	81200:
			TON_DelayTransMove.IN := false;
			IF 	LowerConveyor.InStopped THEN
				tonTimeOut.IN:=FALSE;
				uiExecutingStep:=99000;
			END_IF
			tonTimeOut.IN:=TRUE;
			IF tonTimeOut.Q=TRUE THEN
				strStatus :='Stop conveyor timeout';
				_Error:=TRUE;
			END_IF		
					
    99000: // process done
          Status    := 'Process completed';
      	  _Executed := TRUE;
END_CASE
IF _Executed THEN
    eState := STATE_DONE;
ELSIF _Error THEN
//	FUN_UniqueErrorCodeGenerator(iErrorID := ErrorID,UinqueErrorCode=>_UniqueErrorCode);
    eState := STATE_ERROR;
ELSIF NOT Execute THEN
    eState := STATE_RESETTING;
END_IF
IF _Abort OR Abort THEN
//	FUN_UniqueErrorCodeGenerator(iErrorID := ErrorID,UinqueErrorCode=>_UniqueErrorCode);
	eSTATE:=STATE_ABORTING;
END_IF
END_METHOD

METHOD  M_STATE_RESETTING
VAR_INPUT
END_VAR
Error :=FALSE;
Done :=FALSE;
Busy := FALSE;


CASE uiResettingStep OF
	
	0:
		tonTimeOut.IN:=FALSE;
		TON_DelayTransMove.IN :=FALSE;
		Robot.M_ResetAllCommand();
		Robot.M_ResetRobotAbsMove(TRUE,TRUE);
		uiResettingStep:=100;
		
	100:
	
		LowerConveyor.M_MotorStop();	
		uiResettingStep:=9999;
	9999:
		_ResetCompleted:=TRUE;
END_CASE
IF _ResetCompleted THEN
	eSTATE:=STATE_DORMANT;
END_IF
END_METHOD

END_FUNCTION_BLOCK

// ---- Library/20_MachineUnits/21_StorageArea/Old_version_Service/FB_WareHouseInnerPickToRoundBeltBatch_Old.TcPOU
// ═══════════════════════════════════════════════════════════════════════════
// FB_WareHouseInnerPickToRoundBeltBatch
// 倉儲內層取盒放圓帶 — 批次服務 FB
// ═══════════════════════════════════════════════════════════════════════════
//
// 【用途】
// 管理最多 40 筆「從倉儲內層取盒放上圓帶」流程,每筆由 FB_WareHouseInnerPickToRoundBelt
// 逐筆執行。批次流程由 C# HMI 透過 ADS 寫入 BatchInfo 結構觸發,PLC 端負責
// 驗證資料、迭代處理、handshake 同步動作紀錄給 C#。
//
// 【設計模式】
// 參照 FB_AllocateMoveAutoBatchMode,以「單筆 FB 內嵌 + 批次迭代」架構:
//   1. 收到 Execute → 驗證整批資料安全 (M_ValidateBatchData)
//   2. 迭代 FlowInfo[0..NrOfFlow-1]
//   3. 跳過無效項 (ID = -1 或 A/B 爪皆 NoWork)
//   4. 對每筆有效流程配置並啟動 fbSingleFlow,等其完成/失敗
//   5. 完成後記錄 WorkedID 供 HMI/C# 回報
//   6. 跨迭代 handshake 清理,確保 C# 看到每筆 FeedBack 上升緣
//
// 【FeedBack / ReadComplete 握手協定】(關鍵,跨迭代正確性依賴)
// 每筆 fbSingleFlow 完成時:
//   PLC:   step 99000 → FeedBack := TRUE (通知 C# 陣列可讀)
//   C#:    收到 FeedBack=TRUE → 讀 ActionRecords → set ReadComplete=TRUE
//   PLC:   step 99100 看 ReadComplete=TRUE → 清 FeedBack → 進 DONE
//   C#:    應在看到 FeedBack=FALSE 時清 ReadComplete=FALSE (維持協定)
// 本 Batch FB 為了防 C# 忘記清 ReadComplete 造成下一迭代 skip handshake,
// 在 Step 100 (新迭代開始) 與 Step 300 (迭代結束) 強制清 BatchInfo.ReadComplete。
//
// 【資料安全約束】
// M_ValidateBatchData 在 Step 0 首次進入時呼叫,檢查:
//   - 每個 Work clamp 的 Station 不可為 Undefined
//   - 所有 Work clamp 的 (Station, ReloadCarrier) 不可重複 (同 flow A/B 兩爪也算)
// 違規 → Error + uiResumeStep:=0 (不可續做,需 C# 修正資料重來)
//
// 【Resume / Pause】
// Resume: 錯誤/逾時後 C# 按 Reset → RESETTING 等 fbSingleFlow 回 DORMANT
//         → 若 _bRetry 直接回 EXECUTING 從 uiResumeStep 繼續
//         uiResumeStep 映射固定為 100 (重新配置+啟動 fbSingleFlow),因 abort
//         過程會清掉 fbSingleFlow 內部狀態,不能回原 step 200
// Pause:  僅在「迭代邊界」生效 (step 0 或 310),不中斷單筆流程
//         危險區段 (100~300) 繼續跑到下個邊界才凍結
//
// Create Date : 2026/04/01
// Owner       : Copilot
// ═══════════════════════════════════════════════════════════════════════════

FUNCTION_BLOCK FB_WareHouseInnerPickToRoundBeltBatch_Old EXTENDS FB_ObjectBase_V2 IMPLEMENTS IBasicElement

VAR_INPUT
	// ----- 外部資源參照 (由上層 FB_StorageArea 綁定) -----
	Robot			: REFERENCE TO FB_FanucRobot_Basic_V2;	// 倉儲區 Fanuc 手臂 (取放動作執行者)
	RoundBelt		: REFERENCE TO FB_RoundBeltService;		// 圓帶服務 (目的地,換區偵測)
	WareHouse		: REFERENCE TO FB_WareHouse;				// 倉儲 FB (ReloadBox / FeedInBox)
	Input			: ST_InputTable;						// IO 輸入表 (sensor 等)

	// ----- 批次資料 (C# HMI ↔ PLC 介面) -----
	// BatchInfo 由 C# 透過 ADS 寫入;PLC 讀 FlowInfo[] 並回寫 WorkedID / ActionRecords
	BatchInfo		: REFERENCE TO ST_WareHouseInnerPickBatch;

	Stop			: BOOL;									// 外部停止信號 (DORMANT 時阻擋 Execute 觸發)
END_VAR

VAR_OUTPUT
	// 無額外 output — 完成/錯誤/忙碌狀態透過 BatchInfo.HandShake 回傳 C#
END_VAR

VAR
	// ----- 狀態與錯誤追蹤 -----
	strStatus			: STRING;			// 當前狀態/錯誤描述 (顯示給 HMI)
	tonTimeOut			: TON;				// Per-iteration 逾時計時器 (PT=600s, step 310 推進時重置)
	_UniqueErrorCode	: STRING;			// 錯誤代碼 (E_NOT_AUTO_MODE / E_BATCH_TIMEOUT / E_FLOW_FAILED /
											// E_STATION_UNDEFINED / E_DUPLICATE_TARGET)
	uiResumeStep		: UDINT := 0;		// 續做點步序 (0 = 不可續做, 其他 = RESETTING retry 回此 step)
	_bRetry				: BOOL;				// 續做旗標 (ABORTED → RESETTING → EXECUTING 路徑標記)

	// ----- 批次迭代控制 -----
	iProcessingIndex	: INT := 0;		// 當前處理的流程索引 (0..NrOfFlow-1)
										// 注意: 續做時保留不歸零 (僅 DORMANT 清),保證從中斷點繼續
	CurrentFlow			: ST_WareHouseInnerPickFlowInfo;	// 當前流程資料快取 (避免 C# 改寫中讀取)

	// ----- 內嵌單筆 FB -----
	// 每筆流程都透過這個實例執行;Step 100 配置參照+啟動,Step 310 等其回到 DORMANT
	fbSingleFlow		: FB_WareHouseInnerPickToRoundBelt;
	_bSingleFlowStarted	: BOOL;		// 追蹤 fbSingleFlow 是否有待清理的執行狀態 (用於 ABORTING)
END_VAR

// ============================================================
// 執行順序: input piping → A00 → A10 → output piping
// 讓 state machine 內的 fbSingleFlow() 看到當前 scan 的 C# 輸入
// (ReadComplete),避免 1 scan 延遲
// ============================================================

// 1. Input piping: C# → fbSingleFlow (在 state machine 前)
IF __ISVALIDREF(BatchInfo) THEN
	fbSingleFlow.ReadComplete := BatchInfo.ReadComplete;
END_IF

// 2. Timer PT setup
A00_BasicUnits();

// 3. State machine (含 fbSingleFlow() 呼叫)
SUPER^.A10_StateControl();

// 4. Output piping: fbSingleFlow → C#
IF __ISVALIDREF(BatchInfo) THEN
	BatchInfo.ActionRecords := fbSingleFlow.ActionRecords;
	BatchInfo.ActionIndex := fbSingleFlow.ActionIndex;
	BatchInfo.FeedBack := fbSingleFlow.FeedBack;
	BatchInfo.HandShake.Done := Done;
	BatchInfo.HandShake.Busy := Busy;
	BatchInfo.HandShake.Error := Error;
END_IF
fbSingleFlow (Input := Input);

ACTION A00_BasicUnits:
// 每單筆流程上限 (per-iteration timeout,由 EXECUTING step 310 重置)
// 最多 40 筆 x 600s 單筆 = 6.7hr 批次上限足夠
tonTimeOut(PT := T#900S);
END_ACTION

// 尋找下一筆有效流程
// 從 iProcessingIndex 開始往後掃描 BatchInfo.FlowInfo[]
// 有效條件: ID <> -1 且至少一爪為 Work
// 無效流程自動跳過並記錄 WorkedID
// 回傳 TRUE = 找到有效流程 (iProcessingIndex 已更新), FALSE = 全部完成
METHOD M_FindNextValidFlow : BOOL
VAR_INPUT
END_VAR
VAR
	i		: INT;
	bValid	: BOOL;
END_VAR
IF NOT __ISVALIDREF(BatchInfo) THEN
	M_FindNextValidFlow := FALSE;
	RETURN;
END_IF

IF BatchInfo.NrOfFlow = 0 THEN
	M_FindNextValidFlow := FALSE;
	RETURN;
END_IF

FOR i := iProcessingIndex TO UINT_TO_INT(BatchInfo.NrOfFlow) - 1 BY 1 DO
	bValid := FALSE;

	// 檢查 flow 是否有效 (ID 不為 -1)
	IF BatchInfo.FlowInfo[i].ID <> -1 THEN
		// 檢查是否至少一爪有 Work 行為
		IF BatchInfo.FlowInfo[i].ClampA_Setting.Behavior = E_ClampWork.Work
		OR BatchInfo.FlowInfo[i].ClampB_Setting.Behavior = E_ClampWork.Work THEN
			bValid := TRUE;
		END_IF
	END_IF

	IF bValid THEN
		iProcessingIndex := i;
		CurrentFlow := BatchInfo.FlowInfo[i];
		M_FindNextValidFlow := TRUE;
		RETURN;
	ELSE
		// 標記跳過的 flow 為已處理
		BatchInfo.WorkedID[i] := BatchInfo.FlowInfo[i].ID;
	END_IF
END_FOR

// 沒有更多有效流程
M_FindNextValidFlow := FALSE;
END_METHOD

// ───────────────────────────────────────────────────────────
// M_STATE_ABORTED — 已中止 (可續做錯誤)
// ───────────────────────────────────────────────────────────
// 進入條件:
//   M_STATE_ABORTING 完成清理 (_AbortCompleted=TRUE) 後進入
//
// 特性:
//   - 顯示 Aborted=TRUE + Error=TRUE + strStatus
//   - 等待 C# 透過 BatchInfo.HandShake.Reset 觸發續做或重來
//
// Reset 行為:
//   - uiResumeStep > 0 → 設 _bRetry, uiExecutingStep := uiResumeStep
//                        RESETTING 會等 fbSingleFlow 回 DORMANT 後直接跳 EXECUTING
//                        (從中斷點續做,保留 iProcessingIndex)
//   - uiResumeStep = 0 → 單純 RESETTING → DORMANT,下次 Execute 從頭跑
METHOD M_STATE_ABORTED
VAR_INPUT
END_VAR
Busy := FALSE;
Aborted := TRUE;
Error := TRUE;
Status := strStatus;
_AbortCompleted := FALSE;
uiAbortingStep :=0;

// Support retry/resume on Reset
IF __ISVALIDREF(BatchInfo) THEN
	IF BatchInfo.HandShake.Reset THEN
		IF uiResumeStep > 0 THEN
			uiExecutingStep := uiResumeStep;
			_bRetry := TRUE;
		END_IF
		eState := STATE_RESETTING;
	END_IF
END_IF
END_METHOD

// ───────────────────────────────────────────────────────────
// M_STATE_ABORTING — 中止流程
// ───────────────────────────────────────────────────────────
// 職責:
//   把正在執行的 fbSingleFlow 中止,等其自身 ABORTING → ABORTED
//   跑完後設 _AbortCompleted 進入 STATE_ABORTED。
//   fbSingleFlow 的 ABORTING 內部會處理 Robot/WareHouse/RoundBelt 的資源釋放。
//
// 進入條件:
//   M_STATE_EXECUTING 設 _Abort := TRUE 時觸發
//   (timeout, 單筆流程失敗, Auto mode 脫離等)
//
// 步序:
//   0:    若 _bSingleFlowStarted=TRUE → 發送 fbSingleFlow.Abort := TRUE, 跳 100
//         (若單筆 FB 尚未啟動過,直接跳 9999 略過等待)
//   100:  每 cycle 呼叫 fbSingleFlow() 推進其內部中止狀態機
//         等待條件 (任一滿足): 未啟動 / fbSingleFlow.Aborted / fbSingleFlow 不忙碌
//         → 清 fbSingleFlow.Abort := FALSE, 跳 9999
//   9999: _AbortCompleted := TRUE → base class 轉入 STATE_ABORTED
//
// 注意:
//   iProcessingIndex 不在此清除 (保留供續做),由 DORMANT 才清
METHOD M_STATE_ABORTING
VAR_INPUT
END_VAR
CASE uiAbortingStep OF
0:
	// Abort single-flow FB if running
	IF _bSingleFlowStarted THEN
		fbSingleFlow.Abort := TRUE;
		fbSingleFlow();
	END_IF
	uiAbortingStep := 100;

100:
	// 每 cycle 呼叫 fbSingleFlow() 推進其內部中止狀態機 (ABORTING → ABORTED)
	// 等待條件: 未啟動 / 已中止 / 不在忙碌 → 任一滿足即視為中止完成
	fbSingleFlow();
	IF NOT _bSingleFlowStarted OR fbSingleFlow.Aborted OR NOT fbSingleFlow.Busy THEN
		fbSingleFlow.Abort := FALSE;
		uiAbortingStep := 9999;
	END_IF

9999:
	_AbortCompleted := TRUE;
END_CASE
IF _AbortCompleted THEN
	eState := STATE_Aborted;
END_IF
END_METHOD

// ───────────────────────────────────────────────────────────
// M_STATE_DONE — 批次完成等待
// ───────────────────────────────────────────────────────────
// 批次全部流程成功完成後進入此狀態,設 Done=TRUE 讓 C# 收到完成回報。
// 等 C# 清 BatchInfo.HandShake.Execute (表示收到完成訊號) 後轉 RESETTING。
METHOD M_STATE_DONE
VAR_INPUT
END_VAR
Busy := FALSE;
Done := TRUE;

IF __ISVALIDREF(BatchInfo) THEN
	IF NOT BatchInfo.HandShake.Execute THEN
		eState := STATE_RESETTING;
	END_IF
END_IF
END_METHOD

// ───────────────────────────────────────────────────────────
// M_STATE_DORMANT — 休眠 / 靜止就緒狀態
// ───────────────────────────────────────────────────────────
// 職責:
//   1. 每 scan 重置所有 FB-level 輸出旗標與內部狀態至乾淨初值
//   2. 清除上一輪殘留的 BatchInfo.WorkedID (避免 C# 誤讀舊資料)
//   3. 監聽 BatchInfo.HandShake.Execute / Reset 握手信號
//
// 進入條件:
//   - 從 M_STATE_RESETTING 完成時進入
//   - 首次上電時的初始狀態
//
// 離開條件:
//   - BatchInfo.HandShake.Execute=TRUE AND NOT Stop → STATE_EXECUTING
//
// 備註:
//   每 scan 都跑 (PLC 狀態機性質),所以所有 reset 都必須冪等。
//   M_RecoveryAllObjects 不放這裡,因 fbSingleFlow 的清理由 RESETTING 處理。
METHOD M_STATE_DORMANT
VAR_INPUT
END_VAR
// 清除所有輸出與內部狀態
Busy				:= FALSE;
Done				:= FALSE;
Aborted				:= FALSE;
Error				:= FALSE;
ErrorID				:= 0;
Status				:= '';
_ResetCompleted		:= FALSE;
_Error				:= FALSE;
_Executed			:= FALSE;
_Abort				:= FALSE;
uiExecutingStep		:= 0;
uiResettingStep		:= 0;
uiResumeStep		:= 0;
uiAbortingStep		:= 0;

tonTimeOut.IN		:= FALSE;
_UniqueErrorCode	:= '0';

// 清除批次狀態
iProcessingIndex	:= 0;
_bSingleFlowStarted	:= FALSE;

// 清除上一輪殘留的 WorkedID (避免 C# 誤讀舊資料)
IF __ISVALIDREF(BatchInfo) THEN
	MEMSET(ADR(BatchInfo.WorkedID), 0, SIZEOF(BatchInfo.WorkedID));
END_IF

_AbortCompleted		:= FALSE;
_bRetry				:= FALSE;

// 監聽 HMI/C# 透過 ADS 寫入的 HandShake 信號
// Execute: C# 設定 BatchInfo.HandShake.Execute = TRUE 觸發批次開始
// Reset: C# 在 Error/Aborted 後設定 Reset 清除狀態 (若有 uiResumeStep 則恢復)
IF __ISVALIDREF(BatchInfo) THEN
	IF BatchInfo.HandShake.Execute AND NOT Stop THEN
		Execute := TRUE;
		eState := STATE_EXECUTING;
	END_IF

	IF BatchInfo.HandShake.Reset THEN
		Reset := TRUE;
	END_IF
END_IF
END_METHOD

// ───────────────────────────────────────────────────────────
// M_STATE_ERROR — 不可續做錯誤顯示
// ───────────────────────────────────────────────────────────
// 進入條件:
//   M_STATE_EXECUTING 設 _Error := TRUE (資料驗證失敗等)
//
// 特性:
//   - 此狀態代表「不可續做」,必須 C# 修正資料後從頭重來
//   - 可續做錯誤 (timeout / 單筆失敗) 走 STATE_ABORTING → STATE_ABORTED 路徑
//   - 等 C# 清 BatchInfo.HandShake.Execute 後進 RESETTING
METHOD M_STATE_ERROR
VAR_INPUT
END_VAR
Busy := FALSE;
Error := TRUE;
Status := strStatus;

IF __ISVALIDREF(BatchInfo) THEN
	IF NOT BatchInfo.HandShake.Execute THEN
		eState := STATE_RESETTING;
	END_IF
ELSIF NOT Execute THEN
	eState := STATE_RESETTING;
END_IF
END_METHOD

// ═══════════════════════════════════════════════════════════════════════════
// M_STATE_EXECUTING — 批次迭代執行主狀態
// ═══════════════════════════════════════════════════════════════════════════
//
// 【進入條件】
//   M_STATE_DORMANT 看到 BatchInfo.HandShake.Execute=TRUE AND NOT Stop 後轉入
//
// 【每 cycle 前置檢查】(在 CASE 之前執行)
//   A. Auto mode 檢查: 若不在 Auto → _Abort (避免軸控衝突)
//   B. Pause gate: 僅在 step 0 / 310 (迭代邊界) 生效
//                 危險區段 (100~300) 繼續跑到下個邊界才凍結
//   C. Per-iteration timeout (600s): 超時 → _Abort, uiResumeStep := 100
//
// 【步序總覽】
//   0:      首次進入: M_ValidateBatchData() 整批驗證 (Station 不為 Undefined, 無重複目的地)
//           驗證失敗 → _Error + uiResumeStep:=0 (不可續做)
//           M_FindNextValidFlow(): 從 iProcessingIndex 掃描下一筆有效 flow
//           → 無: 跳 99000 (全部完成)
//           → 找到: 快取 CurrentFlow, 跳 100
//
//   100:    新迭代起始 — 強制清 handshake 狀態 (BatchInfo.FeedBack/ReadComplete + fbSingleFlow.ReadComplete)
//           確保 C# 一定看到本迭代的 FeedBack 上升緣,不被上一迭代的殘留 ack 誤判
//           配置 fbSingleFlow.Robot/RoundBelt/WareHouse/Input/Info/Stop 參照
//           啟動 fbSingleFlow.Execute := TRUE, 跳 200
//
//   200:    等待單筆 FB 完成 — 每 cycle 呼叫 fbSingleFlow() 推進其內部狀態機
//           → fbSingleFlow.Done: 流程成功 → 跳 300
//           → fbSingleFlow.Error/Aborted: 單筆流程失敗 → _Abort,
//             uiResumeStep := 100 (必須回 100 重新配置,因 abort 會清掉 fbSingleFlow 狀態)
//
//   300:    記錄完成 — 寫入 BatchInfo.WorkedID[iProcessingIndex] := CurrentFlow.ID
//           強制清 BatchInfo.ReadComplete (防 C# 遺忘)
//           釋放 fbSingleFlow.Execute := FALSE (讓它進入 RESETTING → DORMANT)
//           跳 310
//
//   310:    等待 fbSingleFlow 完成 RESETTING → DORMANT (Busy/Done/Error 皆 FALSE)
//           避免下一筆配置時與單筆 FB 的清理步序衝突
//           滿足 → iProcessingIndex + 1, 重置 tonTimeOut, 回 0 (處理下一筆)
//
//   99000:  批次全部完成 — _Executed := TRUE → STATE_DONE
//
// 【狀態轉換優先順序】(CASE 後檢查)
//   _Error → STATE_ERROR      (資料驗證失敗等不可續做錯誤)
//   _Abort → STATE_ABORTING   (timeout, 單筆流程失敗等可續做錯誤)
//   _Executed → STATE_DONE    (批次完成)
//
// ═══════════════════════════════════════════════════════════════════════════
METHOD M_STATE_EXECUTING
VAR_INPUT
END_VAR
Busy := TRUE;
tonTimeOut.IN := TRUE;

// 非自動模式直接中止 (避免軸控衝突)
IF GVL_Machine.PackTags[UnitNo.Storage].Status.UnitModeCurrent <> E_UnitMode.Auto THEN
	strStatus := 'Not in Auto mode';
	_UniqueErrorCode := 'E_NOT_AUTO_MODE';
	_Abort := TRUE;
END_IF

// ============================================================
// Pause (Fix P1): 僅在「迭代邊界」生效,避免單筆流程被卡在半途
// 安全 step: 0 (尋找下一筆) / 310 (等 fbSingleFlow 回 DORMANT)
// 危險 step (100~300): 跑完當前這一筆才能凍結
// ============================================================
IF __ISVALIDREF(BatchInfo) AND BatchInfo.Pause THEN
	IF uiExecutingStep = 0 OR uiExecutingStep = 310 THEN
		strStatus := 'Paused (at iteration boundary)';
	END_IF
	// 非安全 step: 繼續跑直到下一個 iteration 邊界
END_IF

// 批次逾時 (per-iteration, step 310 推進時會重置): 單筆上限 600s
// Resume 映射: 無論 timeout 發生在哪個 step,都回 step 100 重新配置 fbSingleFlow
// (abort 過程會清掉 fbSingleFlow 狀態,直接回原 step 沒用)
IF tonTimeOut.Q THEN
	strStatus := 'Batch per-iteration timeout';
	_UniqueErrorCode := 'E_BATCH_TIMEOUT';
	uiResumeStep := 100;
	_Abort := TRUE;
END_IF

CASE uiExecutingStep OF

// ===== Step 0: 資料安全檢查 + 尋找下一筆有效流程 =====
0:
	// 首次進入 (iProcessingIndex=0 且非 retry) 時驗證整個 batch 資料
	// retry 路徑 (_bRetry 由 RESETTING 清) 不重驗,避免重跑時 C# 結構已變
	IF iProcessingIndex = 0 THEN
		IF NOT M_ValidateBatchData() THEN
			// 資料驗證失敗 → 直接報錯,不可續做 (需 C# 修正資料後重來)
			uiResumeStep := 0;
			_Error := TRUE;
			RETURN;
		END_IF
	END_IF

	IF NOT M_FindNextValidFlow() THEN
		// 所有流程已處理完畢 → 跳到完成
		uiExecutingStep := 99000;
	ELSE
		strStatus := CONCAT('Processing flow #', INT_TO_STRING(iProcessingIndex));
		uiExecutingStep := 100;
	END_IF

// ===== Step 100: 配置並啟動單筆 FB =====
100:
	// Safety: 新迭代開始,強制清 handshake 狀態,確保 C# 一定看到本迭代的 FeedBack 上升緣
	// 即使 C# 上一迭代忘了清 ReadComplete,也不會被本迭代的 step 99100 誤認為已 ack
	IF __ISVALIDREF(BatchInfo) THEN
		BatchInfo.FeedBack := FALSE;
		BatchInfo.ReadComplete := FALSE;
	END_IF
	fbSingleFlow.ReadComplete := FALSE;

	// 將手臂/圓帶/倉儲參照及當前流程資料傳入 fbSingleFlow
	fbSingleFlow.Robot REF= Robot;
	fbSingleFlow.RoundBelt REF= RoundBelt;
	fbSingleFlow.WareHouse REF= WareHouse;
	fbSingleFlow.Input := Input;
	fbSingleFlow.Info := CurrentFlow;
	fbSingleFlow.Stop := Stop;
	fbSingleFlow.Execute := TRUE;
	_bSingleFlowStarted := TRUE;
	uiExecutingStep := 200;

// ===== Step 200: 等待單筆 FB 完成 =====
200:
	// 每 cycle 呼叫 fbSingleFlow 推進其狀態機
	fbSingleFlow();

	IF fbSingleFlow.Done THEN
		// 流程成功完成 → 記錄並推進
		uiExecutingStep := 300;
	ELSIF fbSingleFlow.Error OR fbSingleFlow.Aborted THEN
		// 流程失敗 → 中止批次
		// Resume 必須回 step 100 重新配置 fbSingleFlow (abort 後 fbSingleFlow 狀態已被清)
		// 不能回 step 200,因為 step 200 假設 fbSingleFlow 已在執行中
		strStatus := CONCAT('Flow #', CONCAT(INT_TO_STRING(iProcessingIndex), ' failed'));
		_UniqueErrorCode := 'E_FLOW_FAILED';
		uiResumeStep := 100;
		_Abort := TRUE;
	END_IF

// ===== Step 300: 記錄完成 + 釋放單筆 FB =====
300:
	// 寫入 WorkedID 供 HMI/C# 回報
	IF __ISVALIDREF(BatchInfo) THEN
		BatchInfo.WorkedID[iProcessingIndex] := CurrentFlow.ID;
		// Safety: 強制清 C# 的 ack,避免殘留 TRUE 讓下一迭代 skip handshake
		BatchInfo.ReadComplete := FALSE;
	END_IF

	// 釋放單筆 FB: Execute := FALSE → 讓它進入 RESETTING → DORMANT
	fbSingleFlow.Execute := FALSE;
	fbSingleFlow();
	_bSingleFlowStarted := FALSE;
	uiExecutingStep := 310;

// ===== Step 310: 等待單筆 FB 回到 DORMANT 後再推進 =====
310:
	// 確保 fbSingleFlow 完成 RESETTING 流程 (MEMSET + 釋放資源)
	// 避免下一筆流程配置時與 RESETTING 步序衝突
	fbSingleFlow();
	IF NOT fbSingleFlow.Busy AND NOT fbSingleFlow.Done AND NOT fbSingleFlow.Error THEN
		iProcessingIndex := iProcessingIndex + 1;
		// Per-iteration timeout reset: 下一筆重新計時 600s
		tonTimeOut.IN := FALSE;
		uiExecutingStep := 0;
	END_IF

// ===== Step 99000: 批次全部完成 =====
99000:
	_Executed := TRUE;

END_CASE

// ===== 狀態切換 (參照 FB_ObjectBase_V2 / FB_AllocateMoveAutoBatchMode 模式) =====
IF __ISVALIDREF(BatchInfo) THEN
	IF NOT BatchInfo.HandShake.Execute THEN
		eState := STATE_RESETTING;
	ELSIF _Error THEN
		eState := STATE_ERROR;
	ELSIF _Abort THEN
		eState := STATE_ABORTING;
	ELSIF _Executed THEN
		eState := STATE_DONE;
	END_IF
END_IF
END_METHOD

// ───────────────────────────────────────────────────────────
// M_STATE_RESETTING — 重置流程 (含續做分流)
// ───────────────────────────────────────────────────────────
// 職責:
//   從 ABORTED/ERROR/DONE 回到 DORMANT (或直接續做回 EXECUTING),
//   並確保 fbSingleFlow 真的走完自己的 RESETTING → DORMANT,避免 race。
//
// 續做 vs 正常 reset 的差別:
//   - 續做 (_bRetry=TRUE): 由 ABORTED state method 收到 Reset 且 uiResumeStep>0 時設旗標,
//     此時 uiExecutingStep 已被寫回 uiResumeStep (通常是 100),步序 50 等 fbSingleFlow
//     真的回 DORMANT 後,直接跳 STATE_EXECUTING,**不經 DORMANT**,
//     所以 iProcessingIndex 保留、從中斷點繼續。
//   - 正常 reset (_bRetry=FALSE): 步序 50 等 fbSingleFlow 回 DORMANT → 步序 100 → DORMANT,
//     DORMANT 會完整清 iProcessingIndex 等狀態,下次 Execute 從頭跑。
//
// 步序:
//   0:    清 Done/Error/Aborted/tonTimeOut.IN, 下 fbSingleFlow.Reset := TRUE 並呼叫一次
//         無條件跳 50 (無論 _bRetry 真假都要等 fbSingleFlow 真的回 DORMANT)
//   50:   每 cycle 呼叫 fbSingleFlow() 推進其 RESETTING,釋放 Reset
//         等待條件: fbSingleFlow 的 Busy/Done/Error/Aborted 全 FALSE
//         滿足後:
//           _bRetry → 清旗標 + STATE_EXECUTING (續做路徑,跳過 100 與 DORMANT)
//           否則    → 跳 100 (正常路徑)
//   100:  _ResetCompleted := TRUE → base class 轉入 STATE_DORMANT
METHOD M_STATE_RESETTING
VAR_INPUT
END_VAR
CASE uiResettingStep OF
0:
	Done := FALSE;
	Error := FALSE;
	Aborted := FALSE;
	tonTimeOut.IN := FALSE;

	// Reset single-flow FB
	fbSingleFlow.Reset := TRUE;
	fbSingleFlow();

	// _bRetry = TRUE: 由 ABORTED 狀態透過 Reset 觸發
	// 無論 retry 或正常 reset,都要先等 fbSingleFlow 真的回到 DORMANT,
	// 避免 fbSingleFlow 還在 RESETTING 時就被 EXECUTING 視為新迭代
	uiResettingStep := 50;

50:
	// 等待 fbSingleFlow 完成 RESETTING → DORMANT (條件: 所有狀態 flag 都 FALSE)
	fbSingleFlow.Reset := FALSE;
	fbSingleFlow();
	IF NOT fbSingleFlow.Busy AND NOT fbSingleFlow.Done AND NOT fbSingleFlow.Error AND NOT fbSingleFlow.Aborted THEN
		IF _bRetry THEN
			// 續做路徑: uiExecutingStep 已被設回 uiResumeStep,直接回 EXECUTING
			_bRetry := FALSE;
			eState := STATE_EXECUTING;
			RETURN;
		END_IF
		uiResettingStep := 100;
	END_IF

100:
	_ResetCompleted := TRUE;
END_CASE
IF _ResetCompleted THEN 
	eState := STATE_DORMANT;
END_IF
END_METHOD

// 驗證批次資料安全性
// 檢查項目:
//   1. 同一個 (Station, ReloadCarrier) 目的地不能重複出現 (包括同 flow 內 A/B 兩爪)
//   2. 有 Work 的 clamp,其 Station 不能是 Undefined
// 若有任何違規 → 設 Error + strStatus + 回傳 FALSE
// 通過 → 回傳 TRUE
//
// 掃描範圍: BatchInfo.FlowInfo[0..NrOfFlow-1],只檢查 ID<>-1 且 clamp Behavior=Work 的項目
METHOD M_ValidateBatchData : BOOL
VAR_INPUT
END_VAR
VAR
	i, j			: INT;
	nTargets		: INT;					// 已收集的有效目的地數量
	arTargets		: ARRAY[0..79] OF DINT;	// 40 flow x 2 clamp = 80 max. Pack 成 DINT: station*16 + carrier
	nKey			: DINT;
END_VAR
IF NOT __ISVALIDREF(BatchInfo) THEN
	M_ValidateBatchData := FALSE;
	RETURN;
END_IF

nTargets := 0;

FOR i := 0 TO UINT_TO_INT(BatchInfo.NrOfFlow) - 1 BY 1 DO
	IF BatchInfo.FlowInfo[i].ID = -1 THEN
		CONTINUE;
	END_IF

	// ----- A 爪 -----
	IF BatchInfo.FlowInfo[i].ClampA_Setting.Behavior = E_ClampWork.Work THEN
		IF BatchInfo.FlowInfo[i].ClampA_Setting.RoundBeltSetting.Station = E_RoundBeltStation.Undefined THEN
			strStatus := CONCAT('Flow #', CONCAT(INT_TO_STRING(i), ' ClampA Station Undefined'));
			_UniqueErrorCode := 'E_STATION_UNDEFINED';
			M_ValidateBatchData := FALSE;
			RETURN;
		END_IF

		// Pack (Station, ReloadCarrier) → DINT key
		// Station: UINT enum (1..40), Carrier: INT enum (0..4)
		nKey := UINT_TO_DINT(BatchInfo.FlowInfo[i].ClampA_Setting.RoundBeltSetting.Station) * 16
			  + INT_TO_DINT(BatchInfo.FlowInfo[i].ClampA_Setting.RoundBeltSetting.ReloadCarrier);

		// 檢查重複
		FOR j := 0 TO nTargets - 1 BY 1 DO
			IF arTargets[j] = nKey THEN
				strStatus := CONCAT('Duplicate target at flow #', INT_TO_STRING(i));
				_UniqueErrorCode := 'E_DUPLICATE_TARGET';
				M_ValidateBatchData := FALSE;
				RETURN;
			END_IF
		END_FOR
		arTargets[nTargets] := nKey;
		nTargets := nTargets + 1;
	END_IF

	// ----- B 爪 -----
	IF BatchInfo.FlowInfo[i].ClampB_Setting.Behavior = E_ClampWork.Work THEN
		IF BatchInfo.FlowInfo[i].ClampB_Setting.RoundBeltSetting.Station = E_RoundBeltStation.Undefined THEN
			strStatus := CONCAT('Flow #', CONCAT(INT_TO_STRING(i), ' ClampB Station Undefined'));
			_UniqueErrorCode := 'E_STATION_UNDEFINED';
			M_ValidateBatchData := FALSE;
			RETURN;
		END_IF

		nKey := UINT_TO_DINT(BatchInfo.FlowInfo[i].ClampB_Setting.RoundBeltSetting.Station) * 16
			  + INT_TO_DINT(BatchInfo.FlowInfo[i].ClampB_Setting.RoundBeltSetting.ReloadCarrier);

		FOR j := 0 TO nTargets - 1 BY 1 DO
			IF arTargets[j] = nKey THEN
				strStatus := CONCAT('Duplicate target at flow #', INT_TO_STRING(i));
				_UniqueErrorCode := 'E_DUPLICATE_TARGET';
				M_ValidateBatchData := FALSE;
				RETURN;
			END_IF
		END_FOR
		arTargets[nTargets] := nKey;
		nTargets := nTargets + 1;
	END_IF
END_FOR

M_ValidateBatchData := TRUE;
END_METHOD

END_FUNCTION_BLOCK

// ---- Library/20_MachineUnits/21_StorageArea/Service/FB_BoxSupplyCtrl.TcPOU
FUNCTION_BLOCK FB_BoxSupplyCtrl EXTENDS FB_ObjectBase_V2
VAR_INPUT
//    Execute    :BOOL;   // True : This prog will start.
//    Abort      :BOOL;   // True : This prog will be abort.
//    Reset      :BOOL;   // True : This prog will be reset.
//    ObjectName :STRING; // Set this fb name(About it's action)

//	SupplyBTN 				:REFERENCE TO FB_Button;			//2nd machine
//	RackMotor				:REFERENCE TO FB_RackMotor_V2;
//	BoxesPusherCylinder		:REFERENCE TO FB_Cylinder;


	Cylinder				:REFERENCE TO UNI_CylinderList;
	Input 					:REFERENCE TO ST_InputTable;
	Output					:REFERENCE TO ST_OutputTable;
	StroageRegionMode 		:E_UnitMode;
	bAddsBoxRequest 		: BOOL;
	AddBoxes_Status			:ST_AutoAddsBoxesStatus;
	AddBoxes_Ctrl			:ST_AutoAddsBoxesCommand;
	CurrentData 			: ST_SetupPara;
	
END_VAR

VAR_OUTPUT
	RackState : E_RackState;
	AxisRackMotorBTNHomeRequest	:BOOL;
//    Busy    :BOOL;        // True : This prog is running.
//    Done    :BOOL;        // True : Command has been executed.
//    Aborted :BOOL;        // True : This prog is aborted.
//    Error   :BOOL;        // True : This prog has an error.
//    ErrorID :UINT;       // Output ErrorID
//    Status  :T_MaxString; // Output this prog status by string(255bytes)
END_VAR

VAR
//    eState :E_MethodStatus_Basic;
//	uiExecutingStep : UDINT; // This var is used to been controll STATE_EXECUTING process.
//	uiResettingStep : UDINT;
//	uiAbortingStep : UDINT;
//	_Executed :BOOL; // Executing process completed.
//	_Error : BOOL; // FB has an error.
//	_ResetCompleted : BOOL; // FB resetting completed.
//	_AbortCompleted : BOOL; // FB aborting completed.
	RackMotorStationTable   : ARRAY[0..9] OF st_StationPositions;
	uiMaxRackStation :INT :=10;
	_Abort		: BOOL;
	strStatus	: STRING;
	uiResumeStep : UINT;
	ExcutingStep :E_RackState;
	trigBTN			:R_TRIG;
	trigRequest		:R_TRIG;
	tonBtnCtrl		:ton;
	tonBtnMotorCtrl	:ton;
	tonBlinkTimer :TON;
	tonBlink_Internal :TIME :=T#500MS;

END_VAR

A00_BasicUnits();
SUPER^.A10_StateControl();

ACTION A00_BasicUnits:
tonBtnCtrl(PT:=T#5S);
tonBtnMotorCtrl(PT :=T#30S);
ErrorID := 2800;
END_ACTION

METHOD GetModelState
VAR_OUTPUT
    xDone    :BOOL;
    xBusy    :BOOL;
    xError   :BOOL;
    xAborted :BOOL;
    iErrorID :UDINT;
	UniqueErrorCode : STRING;
END_VAR
xDone    := Done;
xBusy    := Busy;
xError   := Error;
xAborted := Abort;
iErrorID := ErrorID;
END_METHOD

METHOD GetName : STRING
GetName := ObjectName;
END_METHOD

METHOD PRIVATE M_Blink : BOOL
VAR_INPUT
	
END_VAR
tonBlinkTimer(IN :=NOT tonBlinkTimer.Q,
				PT := tonBlink_Internal);
IF tonBlinkTimer.Q THEN
	Output.bStorage_StackPushPbLamp := NOT Output.bStorage_StackPushPbLamp;
END_IF
END_METHOD

METHOD PRIVATE M_GetCurrentStation : BOOL
VAR
	i : UINT;
	SetPos	 :LREAL;
END_VAR

VAR_OUTPUT
	uiCurrentStation	:UINT;
END_VAR
//SetPos := THIS^.fbMotor.NcToPlc.SetPos;
SetPos := arAxisCtrl_gb[AxisNo.RackMotor].Admin.Axis.NcToPlc.SetPos;
M_RefreshStationPos();
//IF  THIS^.fbMotor.Status.Homed THEN
IF arAxisCtrl_gb[AxisNo.RackMotor].Admin.Axis.Status.Homed THEN
	FOR i:=0 TO 9 BY 1 DO 
		IF SetPos> RackMotorStationTable[i].Position-5 AND SetPos< RackMotorStationTable[i].Position+5 THEN // Range should be confirm
			uiCurrentStation :=i;
			M_GetCurrentStation :=TRUE;
			RETURN;
		END_IF
	END_FOR
	
	uiCurrentStation:=99;
	M_GetCurrentStation :=FALSE;
ELSE
	M_GetCurrentStation :=FALSE;
	uiCurrentStation:=99;
END_IF
END_METHOD

METHOD PRIVATE M_MoveToStation : BOOL
VAR_INPUT
	uiStation : UINT;
END_VAR
VAR
	bDone	:BOOL;
	uiTargetPosition	:LREAL ;
END_VAR
M_RefreshStationPos();
IF uiStation>=0 AND uiStation <10 THEN
	uiTargetPosition :=RackMotorStationTable[uiStation].Position;
	
	arAxisCtrl_gb[AxisNo.RackMotor].PosMode.Acc := CurrentData.Axes.RackMotor.HalfAuto.Acceleration;
	arAxisCtrl_gb[AxisNo.RackMotor].PosMode.Dec := CurrentData.Axes.RackMotor.HalfAuto.Deceleration;
	arAxisCtrl_gb[AxisNo.RackMotor].PosMode.Jerk := CurrentData.Axes.RackMotor.HalfAuto.Jerk;
	arAxisCtrl_gb[AxisNo.RackMotor].PosMode.Velocity := CurrentData.Axes.RackMotor.HalfAuto.Velocity;
	arAxisCtrl_gb[AxisNo.RackMotor].PosMode.Position := uiTargetPosition;
	
//	THIS^.fbMotor.MoveAbs(lrPosition	:=uiTargetPosition,
//						lrVelocity 		:=GVL.MotorCore[AxisNo.RackMotor].VCC,
//						lrAcceleration	:=GVL.MotorCore[AxisNo.RackMotor].ACC,
//						lrDeceleration	:=GVL.MotorCore[AxisNo.RackMotor].DCC,
//						lrJerk			:=GVL.MotorCore[AxisNo.RackMotor].Jerk,
//						BufferMode		:=MC_BufferMode.MC_Aborting);
	//THIS^.fbMotor.GetCmdDoneStatus(bMotionCmdDone=>bDone);
ELSE
	M_MoveToStation :=FALSE;
	RETURN;
END_IF
END_METHOD

METHOD PRIVATE M_RefreshStationPos : BOOL
VAR_INPUT
END_VAR
VAR
	i: UINT;
	position : ST_PositionTable;
END_VAR
FOR i := 0 TO 9 DO
	position :=FUN_GetPositionTableData(PositionName:='W',Index:=i,Clip:=0);
RackMotorStationTable[i].Position:= position.X_Pos;
END_FOR
	M_RefreshStationPos :=TRUE;

// todo : update position of each stations
//FOR i:=1 TO 200 BY 1 DO
//	FOR iIndex:=0 TO 9 BY 1 DO
//		IF 		
//			DAS_CoreSys.MachineControl.CurrentData.PositionTable[i].Index= iIndex AND
//			DAS_CoreSys.MachineControl.CurrentData.PositionTable[i].Zone ='W' THEN
//			RackMotorStationTable[iIndex].Position := DAS_CoreSys.MachineControl.CurrentData.PositionTable[i].X_Pos;

//			StationsPosition[iIndex]:=RackMotorStationTable[i].Position;
//		ELSE
//			M_RefreshStationPos :=FALSE;
//		END_IF
//	END_FOR
//END_FOR
END_METHOD

METHOD  M_STATE_ABORTED
VAR_INPUT
END_VAR
ERROR :=TRUE;
Busy    := FALSE;
Aborted := TRUE;
Status := strStatus;

IF NOT Execute THEN
	eSTATE:=STATE_RESETTING;
END_IF

IF Execute AND Reset THEN
	uiExecutingStep :=uiResumeStep;
	eSTATE:=STATE_EXECUTING;
END_IF
END_METHOD

METHOD  M_STATE_ABORTING
VAR_INPUT
END_VAR
CASE uiAbortingStep OF
	0 :
		uiAbortingStep:=9999;
	
	9999:	_AbortCompleted:=TRUE;
END_CASE

IF _AbortCompleted THEN	
	eSTATE :=STATE_ABORTED;
END_IF
END_METHOD

METHOD  M_STATE_DONE
VAR_INPUT
END_VAR
Busy 	:= FALSE;
Done	:=TRUE;

IF NOT Execute THEN
	eSTATE:=STATE_RESETTING;
END_IF
END_METHOD

METHOD  M_STATE_DORMANT
VAR_INPUT
END_VAR
Busy            := FALSE;
Done            := FALSE;
Aborted         := FALSE;
Error           := FALSE;
ErrorID         := 0;
Status          := '';
_ResetCompleted := FALSE;
_Error          := FALSE;
_Executed       := FALSE;
strStatus :='FB_BoxSupplyCtrl: No Error';
uiExecutingStep :=uiResettingStep :=uiResumeStep :=0;

IF Execute THEN
	eSTATE:=STATE_EXECUTING;
END_IF
END_METHOD

METHOD  M_STATE_ERROR
VAR_INPUT
END_VAR
ERROR   :=TRUE;
Busy	:=FALSE;
Status := strStatus;
M_TurnOff();
RackState:= E_RackState.idle; // Useless so far
AxisRackMotorBTNHomeRequest :=false;
IF NOT Execute OR Reset THEN // Execute will always on , therefor Reset is only way to recovery from error	
	eSTATE:=STATE_RESETTING;
END_IF
END_METHOD

METHOD  M_STATE_EXECUTING
VAR_INPUT
END_VAR

VAR_INST
	uiTransitingStep : UINT;
	uiTargetStation :UINT :=0;
	bFreeState	  :BOOL;
END_VAR

VAR
	bMotionDone			:BOOL;
	_uiCurrentStation	:UINT;
END_VAR
Busy :=TRUE;	
//IF SupplyBTN.P_IsBTNRef THEN			//2nd machine 
//	trigBTN(CLK:= (SupplyBTN.P_ButtonState));
//END_IF //Make sure BTN is referenced otherwise exception occur

	trigBTN(CLK:= ( Input.bStorage_StackPushPb));
trigRequest(CLK :=(AddBoxes_Status.InterventionRequest AND bFreeState));

// Force state control
IF AddBoxes_Status.Busy OR AddBoxes_Status.Done  THEN	
	ExcutingStep := E_RackState.AddBoxes;
	
ELSIF StroageRegionMode = E_UnitMode.MANUAL AND
	arAxisCtrl_gb[AxisNo.RackMotor].Admin.Axis.Status.HasJob AND
//	  rackmotor.fbMotor.Status.HasJob AND 
	  NOT (ExcutingStep = E_RackState.FeedBox) THEN	
			ExcutingStep := E_RackState.ManualCtrl;

ELSIF	StroageRegionMode = E_UnitMode.MANUAL AND 
		NOT Cylinder.List.fbStackPush.InRearPosition AND
//		BoxesPusherCylinder.P_IsMoving AND 
		NOT	(ExcutingStep = E_RackState.FeedBox) THEN	
			ExcutingStep := E_RackState.ManualCtrl;

			
END_IF

RackState := ExcutingStep;

CASE ExcutingStep OF
	

	E_RackState.idle:
		;	
	E_RackState.AddBoxes:
		//Service AddBox working
		M_TurnOff();
		bFreeState:=FALSE;
		IF NOT AddBoxes_Ctrl.Execute AND NOT AddBoxes_Status.Error  THEN
        	ExcutingStep := E_RackState.Free;
    	END_IF
		
	E_RackState.ManualCtrl:
	//Stroage area in manual and Rack is moving
		M_TurnOff();
		bFreeState:=FALSE;
		IF NOT arAxisCtrl_gb[AxisNo.RackMotor].Admin.Axis.Status.HasJob AND Cylinder.List.fbStackPush.InRearPosition THEN
            ExcutingStep := E_RackState.Free;
        END_IF
		
	E_RackState.FeedBox:
	// FeedBox mode , 
		M_Blink();
		bFreeState:=FALSE;
		AxisRackMotorBTNHomeRequest :=false;
			IF	trigBTN.Q THEN				
				ExcutingStep :=E_RackState.TransitingFree;	
			END_IF
			
	E_RackState.Free:
	// Rack is free , User is allow to ask to suply box by push the suplyBTN
		M_TurnOn();
		bFreeState:=TRUE;
			 IF trigBTN.Q OR trigRequest.Q THEN
				 uiTransitingStep:=0;
				 ExcutingStep := E_RackState.TransitingFeedBox;
			 END_IF

	E_RackState.TransitingFree:
			 IF NOT AddBoxes_Status.InterventionRequest THEN
				 ExcutingStep :=E_RackState.Free;	
			 END_IF
		
	E_RackState.TransitingFeedBox:
	//Transition step , from Free to FeedBox
		//M_Blink();
		M_TurnOff();
		bFreeState:=FALSE;
		AxisRackMotorBTNHomeRequest :=TRUE;
		// todo : if transition step needs different indication of BTN behavior?
		CASE uiTransitingStep OF
		0:
			tonBtnCtrl.IN	:=FALSE;
			tonBtnMotorCtrl.IN :=FALSE;
			uiTransitingStep:=5;
			M_GetCurrentStation(uiCurrentStation =>_uiCurrentStation);
			IF uiTargetStation = _uiCurrentStation THEN
				uiTransitingStep :=30;
			END_IF
			
		5:	//Move cylinder back
			tonBtnCtrl.IN:=TRUE;			
			Cylinder.List.fbStackPush.M_Retract();
			IF Cylinder.List.fbStackPush.InRearPosition AND NOT arAxisCtrl_gb[AxisNo.RackMotor].Admin.Axis.Status.HasJob THEN 
				tonBtnCtrl.IN :=FALSE;
				uiTransitingStep :=10;
			END_IF
			IF tonBtnCtrl.Q THEN
				_Error:= TRUE;
				StrStatus :='FB_BoxSupplyCtrl Step 5: Cylinder MoveBackward timeout';
			END_IF
		10:	// Rackmotor move to station 0
			tonBtnMotorCtrl.IN :=TRUE;
			M_MoveToStation(uiTargetStation);
			IF arAxisCtrl_gb[AxisNo.RackMotor].Admin.Axis.Status.HasJob THEN
				tonBtnMotorCtrl.IN :=FALSE;
			uiTransitingStep :=20;
			END_IF
			IF tonBtnMotorCtrl.Q THEN
				_Error :=TRUE;
				StrStatus :='FB_BoxSupplyCtrl Step 10: RackMotor MoveToStation timeout';
			END_IF
		20:	// check currentstation 
			tonBtnMotorCtrl.IN :=TRUE;
//			bMotionDone :=rackmotor.fbMotor.Status.InTargetPosition;
			bMotionDone :=arAxisCtrl_gb[AxisNo.RackMotor].Admin.Axis.Status.InTargetPosition;
			M_GetCurrentStation(uiCurrentStation =>_uiCurrentStation);
			IF bMotionDone  AND uiTargetStation = _uiCurrentStation THEN
				
				uiTransitingStep :=30;
			END_IF
			IF tonBtnMotorCtrl.Q THEN
				_Error :=TRUE;
				StrStatus :='FB_BoxSupplyCtrl Step 20: RackMotor currentStation timeout';
			END_IF
		30:
			tonBtnMotorCtrl.IN :=FALSE;
			ExcutingStep := E_RackState.FeedBox;
			AxisRackMotorBTNHomeRequest :=FALSE;
		END_CASE
		


END_CASE
	
IF NOT Execute THEN
	eState:=STATE_RESETTING;
END_IF
IF _Error THEN
	eState:=STATE_ERROR;
END_IF
IF _Abort THEN
	eSTATE:=STATE_ABORTING;
END_IF
IF _Executed THEN
	eSTATE:=STATE_Done;
END_IF
END_METHOD

METHOD  M_STATE_RESETTING
VAR_INPUT
END_VAR
Error :=FALSE;
Done :=FALSE;
Busy := FALSE;
AxisRackMotorBTNHomeRequest :=FALSE;
tonBtnCtrl.IN := FALSE;
tonBtnMotorCtrl.IN := FALSE;
M_TurnOff();
CASE uiResettingStep OF
	
	0:
		uiResettingStep:=9999;


	9999:
		_ResetCompleted:=TRUE;
END_CASE
IF _ResetCompleted THEN
	eSTATE:=STATE_DORMANT;
END_IF
END_METHOD

METHOD PRIVATE M_TurnOff : BOOL
VAR_INPUT
END_VAR
Output.bStorage_StackPushPbLamp := false;
END_METHOD

METHOD PRIVATE M_TurnOn : BOOL
VAR_INPUT
END_VAR
Output.bStorage_StackPushPbLamp := true;
END_METHOD

END_FUNCTION_BLOCK

// ---- Library/20_MachineUnits/21_StorageArea/Service/FB_LowerFeedInConveyor.TcPOU
FUNCTION_BLOCK FB_LowerFeedInConveyor EXTENDS FB_ActionBasic
VAR_INPUT
    xExecute    : BOOL;
    xAbort      : BOOL;
	xReset		: BOOL;
    Cylinder 	: REFERENCE TO UNI_CylinderList;
    TimeOut  	: LREAL := 30; // Unit : s
	Input		: ST_InputTable;
	OutPut		: ST_OutputTable;
	Motor		: REFERENCE TO UNI_MotorList;
END_VAR	
VAR_OUTPUT
    xAborted : BOOL;
    iErrorID : INT;
    ErrorMsg : T_MaxString;
END_VAR
VAR
    StateBehaviour   : CBML.ETrigATo;
    CurrentPosition : ST_PositionTable;
	uiCyclicStep    : UINT := 0;
	Reset_Rtrig 	:R_TRIG;
	
	TON_SensorDelay :TON;
	TON_ArrivedTimeOut :TON;
	TON_TimeOut :TON;
	fbExecuteEdgeDetect :FB_EdgeDetect;
END_VAR

THIS^.IBehaviourModel := StateBehaviour;
StateBehaviour(xExecute := xExecute,
              xAbort := xAbort OR fbExecuteEdgeDetect.xFallingEdge,
              udiTimeOut := LREAL_TO_UDINT( TimeOut*1000000),
              xDone => xDone,
              xBusy => xBusy,
              xError => xError,
              xAborted => xAborted);
//Error Mes
iErrorID := StateBehaviour._model.iErrorID;
ErrorMsg := M_GetErrorMsg(xErrorID := iErrorID);  

//Make sure that C# turns off execute to shut down the service
fbExecuteEdgeDetect(xInput :=xExecute);

//Reset 
Reset_Rtrig(CLK:= xReset);
IF Reset_Rtrig.Q THEN
	StateBehaviour.ResetModel(xCommit:=xReset);
END_IF

//Action
A00_BaseUnits();

ACTION A00_BaseUnits:
TON_SensorDelay(PT:= T#500MS);
TON_ArrivedTimeOut(PT:=T#30S);
TON_TimeOut(PT:=T#10S);
END_ACTION

METHOD CleanupAction
VAR_INPUT
    xAbortProposed : BOOL;
    iErrorIDProposed: INT;
END_VAR
VAR_OUTPUT
    xComplete : BOOL := TRUE;
    xAbort: BOOL := xAbortProposed;
 	iErrorID : INT := iErrorIDProposed;
END_VAR
END_METHOD

METHOD CyclicAction
VAR_INPUT
    itfTimingController : CBML.ITimingController;
END_VAR
VAR_OUTPUT
    xComplete : BOOL := TRUE;
    iErrorID : INT := 0;
END_VAR
xComplete :=FALSE;

CASE uiCyclicStep OF 
	
	100:	//檔盒上升， 呼叫輸送帶
		TON_TimeOut.IN:= TRUE;
		Cylinder.List.fbLowCV_Block2.M_Extend();
		IF Cylinder.List.fbLowCV_Block2.InFrontPosition THEN
			TON_TimeOut.IN:=FALSE;
			Motor.List.LowCV.M_MoveForward();
			uiCyclicStep:=150;
		END_IF
		IF TON_TimeOut.Q THEN 
			iErrorID :=10;
		END_IF
	150:	//check motor forward
		TON_TimeOut.IN :=TRUE;
		IF Motor.List.LowCV.InForWard THEN 
			TON_TimeOut.IN:=FALSE;
			uiCyclicStep:=200;
		END_IF
		IF TON_TimeOut.Q THEN
			iErrorID :=11;
		END_IF
	
	200:	//盒子到位, 延遲訊號,
		TON_ArrivedTimeOut.IN:= TRUE;
		TON_SensorDelay.IN := Input.bLowCV_Block2Detect_Sensor;
		IF TON_SensorDelay.Q THEN
			TON_SensorDelay.IN:=FALSE;
			TON_ArrivedTimeOut.IN:=FALSE;
			Cylinder.List.fbLowCV_Press4.M_Extend();
			uiCyclicStep:=300;
		END_IF
		IF TON_ArrivedTimeOut.Q THEN
			iErrorID :=9;
		END_IF
		
	300:	//檔盒下 等待第一盒到達最前sensor
		TON_TimeOut.IN:=TRUE;
		IF Cylinder.List.fbLowCV_Press4.InFrontPosition THEN
			Cylinder.List.fbLowCV_Block2.M_Retract();
		END_IF
		IF Cylinder.List.fbLowCV_Block2.InRearPosition THEN
			TON_TimeOut.IN:=FALSE;
			uiCyclicStep:=400;	
		END_IF
		IF TON_TimeOut.Q THEN
			iErrorID :=11;
		END_IF
		
	400:	//確認到最前sensor 
		TON_SensorDelay.IN:=Input.bLowCV_BoxArrived_Sensor;
		IF TON_SensorDelay.Q THEN
			TON_SensorDelay.IN:=FALSE;
			Cylinder.List.fbLowCV_Block2.M_Extend();
			uiCyclicStep:=500;
		END_IF
	
	500:	//釋放第二盒 
		IF 	Cylinder.List.fbLowCV_Block2.InFrontPosition THEN
			Cylinder.List.fbLowCV_Press4.M_Retract();
			uiCyclicStep:=600;
		END_IF
	600:	// 第二盒到檔盒位 第三盒壓盒檔上
		TON_SensorDelay.IN:= Input.bLowCV_Block2Detect_Sensor;
		IF TON_SensorDelay.Q THEN
			TON_SensorDelay.IN :=FALSE;
			Cylinder.List.fbLowCV_Press4.M_Extend();
			uiCyclicStep:= 700;
		END_IF
	
	700:	//釋放第二盒
		IF Cylinder.List.fbLowCV_Press4.InFrontPosition THEN
			Cylinder.List.fbLowCV_Block2.M_Retract();
			Cylinder.List.fbLowCV_Block1.M_Extend();
		END_IF
		IF Cylinder.List.fbLowCV_Block2.InRearPosition AND 
			Cylinder.List.fbLowCV_Block1.InFrontPosition THEN
			uiCyclicStep:= 800;
		END_IF
		
	800:	// 等待第二盒到夾盒位
		TON_SensorDelay.IN:=Input.bLowCV_Block1Detect_Sensor;
		IF TON_SensorDelay.Q THEN
			TON_SensorDelay.IN:=FALSE;
			Motor.List.LowCV.M_MotorStop();
			uiCyclicStep:=900;
		END_IF
	900:	//馬達停止 第一第二盒壓盒上
		IF Motor.List.LowCV.InStopped THEN
			Cylinder.List.fbLowCV_Press1.M_Extend();
			Cylinder.List.fbLowCV_Press2.M_Extend();
			Cylinder.List.fbLowCV_Block1.M_Retract();
			uiCyclicStep :=1000;
		END_IF
	1000:	//壓盒下
		IF Cylinder.List.fbLowCV_Press1.InFrontPosition AND 
			Cylinder.List.fbLowCV_Press2.InFrontPosition AND 
			Cylinder.List.fbLowCV_Block1.InRearPosition THEN
			Cylinder.List.fbLowCV_Press1.M_Retract();
			Cylinder.List.fbLowCV_Press2.M_Retract();
		END_IF
	1100:	//確認壓盒位置 回done
		IF Cylinder.List.fbLowCV_Press1.InRearPosition AND 
			Cylinder.List.fbLowCV_Press2.InRearPosition THEN 
			xComplete :=TRUE;
		END_IF
END_CASE
END_METHOD

METHOD ExitAction
VAR_INPUT
    xAfterCleanup : BOOL;
    xInCopyCode : BOOL;
END_VAR
TON_SensorDelay.IN:=FALSE;
END_METHOD

METHOD M_GetErrorMsg : T_MaxString
VAR_INPUT
	xErrorID: INT;
END_VAR

VAR
	
END_VAR
CASE xErrorID OF
	0:
		M_GetErrorMsg := 'No Error';
	1:
		M_GetErrorMsg := 'FB_LowerFeedInConveyor ErrorID 1: Action time out';
	2:
		M_GetErrorMsg := 'FB_LowerFeedInConveyor ErrorID 2: Position Data invalid';
	3:
		M_GetErrorMsg := 'FB_LowerFeedInConveyor ErrorID 3: LowCV_Block1 has Error in StartAction ';
	4:
		M_GetErrorMsg := 'FB_LowerFeedInConveyor ErrorID 4: LowCV_Block2 has Error in StartAction';
	5:
		M_GetErrorMsg := 'FB_LowerFeedInConveyor ErrorID 5: LowCV_Press1 has Error in StartAction';
	6:
		M_GetErrorMsg := 'FB_LowerFeedInConveyor ErrorID 6: LowCV_Press2 has Error in StartAction';
	7:
		M_GetErrorMsg := 'FB_LowerFeedInConveyor ErrorID 7: fbLowCV_Press3 has Error in StartAction';
	8:
		M_GetErrorMsg := 'FB_LowerFeedInConveyor ErrorID 8: fbLowCV_Press4 has Error in StartAction';
	9:
		M_GetErrorMsg := 'FB_LowerFeedInConveyor ErrorID 9: Box Arrived Time out not on LowCVBlock2' ;
	10:
		M_GetErrorMsg := 'FB_LowerFeedInConveyor ErrorID 10: Cylinder Error in CyclicAction';
	11:
		M_GetErrorMsg := 'FB_LowerFeedInConveyor ErrorID 11: Motor Error in CyclicAction';
									
		
		
		
		
END_CASE
END_METHOD

METHOD ResetAction
VAR_OUTPUT
    xComplete : BOOL := TRUE;
END_VAR
END_METHOD

METHOD StartAction
VAR_OUTPUT
    xComplete : BOOL := TRUE;
	iErrorID : INT := 0;
END_VAR
xComplete :=FALSE;

TON_SensorDelay.IN:=FALSE;

IF Cylinder.List.fbLowCV_Block1.xError THEN
	iErrorID := 3;
END_IF
IF Cylinder.List.fbLowCV_Block2.xError THEN
	iErrorID := 4;
END_IF
IF Cylinder.List.fbLowCV_Press1.xError THEN
	iErrorID := 5;
END_IF
IF Cylinder.List.fbLowCV_Press2.xError THEN
	iErrorID := 6;
END_IF
IF Cylinder.List.fbLowCV_Press3.xError THEN
	iErrorID := 7;
END_IF
IF Cylinder.List.fbLowCV_Press4.xError THEN
	iErrorID := 8;
END_IF

IF Cylinder.List.fbLowCV_Block1.InRearPosition AND
	Cylinder.List.fbLowCV_Block2.InRearPosition AND 
	Cylinder.List.fbLowCV_Press1.InRearPosition AND 
	Cylinder.List.fbLowCV_Press2.InRearPosition AND 
	Cylinder.List.fbLowCV_Press3.InRearPosition AND 
	Cylinder.List.fbLowCV_Press4.InRearPosition AND 
	Input.bLowCV_2ndBoxGap_Sensor THEN	//reverse logic sensor ,do make sure no box here 
	xComplete :=TRUE;
END_IF
END_METHOD

END_FUNCTION_BLOCK

// ---- Library/20_MachineUnits/22_AllocateArea/Old_Version_Service/FB_AllocateMoveAutoBatchMode_Reverse_Old.TcPOU
FUNCTION_BLOCK FB_AllocateMoveAutoBatchMode_Reverse_Old EXTENDS FB_ObjectBase_V2
VAR_INPUT
//    Execute    :BOOL;   // True : This prog will start.
//    Abort      :BOOL;   // True : This prog will be abort.
//    Reset      :BOOL;   // True : This prog will be reset.
//    ObjectName :STRING; // Set this fb name(About it's action)
//	Pause				:BOOL;
	bOccupied			: BOOL;	
	Clips 				: REFERENCE TO  ARRAY[0..3] OF FB_Cylinder;
	cylinders 			: REFERENCE TO  ARRAY[0..3] OF FB_Cylinder;	
	TurnTable_Press		 		   : REFERENCE TO FB_Cylinder;
	RoundBelt_Press 			   : REFERENCE TO FB_Cylinder;
	AutoAllocateJobBatch_Reverse_Ctrl      :st_AllocateMoveAutoBatchMode_Ctrl;
	INPUT            			   : REFERENCE TO ST_InputTable;
    OUTPUT           			   : REFERENCE TO ST_OutputTable;
	NrOfAllocateCylinder 		   : INT :=4;
	CurrentData 				   : REFERENCE TO ST_SetupPara; // Componets setup parameter
	bAutoAllocateJobDryRun         : BOOL := FALSE;
	RoundBeltMoveJob_Status 		: ST_StatusBasic;
END_VAR

VAR_OUTPUT
//    Busy    :BOOL;        // True : This prog is running.
//    Done    :BOOL;        // True : Command has been executed.
//    Aborted :BOOL;        // True : This prog is aborted.
//    Error   :BOOL;        // True : This prog has an error.
//    ErrorID :UINT;       // Output ErrorID
//    Status  :T_MaxString; // Output this prog status by string(255bytes)
	RoundBeltMoveJob_Ctrl : ST_CommandBasic;
	ProcessedIndex : ARRAY[0..49] OF INT;
	//UniqueErrorCode :STRING;
	// AutoAllocateJobBatch_Status    :st_AllocateMoveAutoBatchMode_Status;
	RoundBeltMoveJob_Position	:LREAL;
	bAllocateRobotMoveRequest	: BOOL;
END_VAR

VAR
//    eState :E_MethodStatus_Basic;
//	uiExecutingStep : UDINT; // This var is used to been controll STATE_EXECUTING process.
//	uiResettingStep : UDINT;
//	uiAbortingStep : UDINT;
//	_Executed :BOOL; // Executing process completed.
//	_Error : BOOL; // FB has an error.
//	_ResetCompleted : BOOL; // FB resetting completed.
//	_AbortCompleted : BOOL; // FB aborting completed.
//	_Abort		: BOOL;
	strStatus	: STRING;
	uiResumeStep : UINT;

//	bSimpleAllocationBatchEnable		 :BOOL;
//	AutoRotatebelt_Internal_Ctrl   : st_RoundBeltAutoSingleMove_Ctrl;
	_UniqueErrorCode : STRING;
	arrProcessedIndex : ARRAY[0..49] OF INT;
 //   eState              :E_MethodStatus_Basic;  
  //  uiAbortingStep      :UDINT;
    uiAbortedStep       :UDINT;
  //  uiResettingStep     :UDINT;
	uiResumableStep		: E_AllocationJob;
    bAborttingCompleted :BOOL; // True: Aborting process finished
    bAborted            :BOOL; // True : Aborted process finished
    bExecuted           :BOOL; // True : Executing process finished
    bResettingCompleted :BOOL; // True : Resetting process finished  
    iWorkingIndex		:UINT:=0;	
	iProcessingIndex	:INT :=0;
	iWorkingCylinder	:INT;
	//_Error				:BOOL :=FALSE;
	StatusDescription	:STRING;
	ClipsHaveNeedle		: ARRAY[0..3] OF BOOL;
	ClipsHaveNeedle_Pick		: ARRAY[0..3] OF BOOL;
	ClipsHaveNoNeedle	: ARRAY[0..3] OF BOOL;
	bCylinderCheck 		: BOOL;
	bCylinderCheckFastMode : BOOL;
	iPickingNeedleCount		:INT;
	iPlacingNeedleCount		:INT;
	bIfNextCycle			:BOOL;
	bCheckStation			:BOOL:=FALSE;
	
	
	
	tAutoAllocationJobBatchTimeOut_Reverse:Tc2_Standard.TON;
    sAllocationJobBatchStatus      :STRING;
    tonFastModeTimeDelayBatch_Reverse      :Tc2_Standard.TON;
	AllocationJobBatchModeReverse		:E_AllocationJob := E_AllocationJob.Defult;
	 Ton_RoundBeltArrivedDelay     : TON;
	 CurrentPosition : ST_PositionTable;
	
  	RoundBeltMoveJob : st_AllocateCircleMoveStructure;	
		
//==========================M_AllocationJobBatchMode================================

	{attribute 'hide'}
	bCheckTrue : BOOL:=TRUE;
	iCurrentRotateBeltStation : UINT;
	i : UINT;	
	j : UINT;	

	bMoveRotateBeltBusy	:BOOL;
	bMoveRotateBeltDone : BOOL;
	A1Used				:BOOL :=FALSE;
	A2Used				:BOOL :=FALSE;
	R1Used				:BOOL :=FALSE;
	R2Used				:BOOL :=FALSE;
	bBoxCheck			:BOOL :=TRUE;
	PickingStation		:UINT;
	iNextPickingStation :UINT;
	
	

	
	
END_VAR

A00_BasicUnits();
SUPER^.A10_StateControl();

(*============================================================
Create Date : 2026/04/27	
Last Update	: 2026/04/27
Change Log  : 將此版本封版，導入鏡射機測試完成版本。 edited by Gamin 
============================================================*)

ACTION A00_BasicUnits:
Ton_RoundBeltArrivedDelay();
tonFastModeTimeDelayBatch_Reverse(PT:=T#100MS);
tAutoAllocationJobBatchTimeOut_Reverse(PT:=T#30s);
END_ACTION

METHOD GetModelState
VAR_OUTPUT
    xDone    :BOOL;
    xBusy    :BOOL;
    xError   :BOOL;
    xAborted :BOOL;
    iErrorID :UDINT;
	UniqueErrorCode : STRING;
END_VAR
xDone    := Done;
xBusy    := Busy;
xError   := Error;
xAborted := Abort;
iErrorID := ErrorID;
END_METHOD

METHOD GetName : STRING
GetName := ObjectName;
END_METHOD

(* Check Allocate Robot Clip cylinder no error
	Return True : no error
*)
METHOD M_CheckClipsNoError : BOOL
VAR_INPUT
END_VAR
//IF Clips[E_ClipsNo.ClipA].bError OR Clips[E_ClipsNo.ClipB].bError OR Clips[E_ClipsNo.ClipC].bError OR Clips[E_ClipsNo.ClipD].bError THEN
//    M_CheckClipsNoError := FALSE;
//ELSE
//    M_CheckClipsNoError := TRUE;
//END_IF
M_CheckClipsNoError := TRUE;
END_METHOD

(* Check Allocate Robot vertical cylinder no error
	return True : no error
*)
METHOD M_CheckCylindersNoError : BOOL
VAR_INPUT
END_VAR
//IF cylinders[E_CylinderNo.CylinderA].bError OR
//   cylinders[E_CylinderNo.CylinderB].bError OR
//   cylinders[E_CylinderNo.CylinderC].bError OR
//   cylinders[E_CylinderNo.CylinderD].bError
//THEN
//    M_CheckCylindersNoError := FALSE;
//ELSE
//    M_CheckCylindersNoError := TRUE;
//END_IF

M_CheckCylindersNoError := TRUE;
END_METHOD

METHOD PRIVATE M_RecoveryAxes : BOOL
VAR_INPUT
END_VAR
VAR
	bCheckTrue : BOOL;
	CheckErrorIndex : UINT;
END_VAR
bCheckTrue := TRUE;
FOR CheckErrorIndex:=1 TO 4 DO 
	IF arAxisCtrl_gb[CheckErrorIndex].Admin.Axis.Status.Error THEN
		arAxisCtrl_gb[CheckErrorIndex].Admin.ClearError:=TRUE;
		bCheckTrue:=FALSE;
	ELSE
		arAxisCtrl_gb[CheckErrorIndex].Admin.ClearError:=FALSE;	
	END_IF
END_FOR
//		TurnTable := 1,
//      RoundBelt := 2,
//      Allocate_X := 3,
//      Allocate_Y := 4,

M_RecoveryAxes:= bCheckTrue;
END_METHOD

METHOD  M_STATE_ABORTED
VAR_INPUT
END_VAR
Busy     := FALSE;
Aborted := TRUE;
Status                       := StatusDescription;
Error                        := TRUE;

IF Aborted AND NOT Execute THEN
    eState := STATE_RESETTING;
END_IF

	ErrorID						 := 108;

IF Aborted AND Reset THEN
	AllocationJobBatchModeReverse :=uiResumableStep;
	eState :=STATE_EXECUTING;
	Aborted :=FALSE;
END_IF
END_METHOD

METHOD  M_STATE_ABORTING
VAR_INPUT
END_VAR
CASE uiAbortingStep OF
            0:
				tAutoAllocationJobBatchTimeOut_Reverse.IN:=FALSE;
				
				uiAbortingStep:=100;
                // Aborting process start
                
			100:
//					FOR i:=1 TO GVL.NrOfAllocateCylinder DO
					
//					IF  clips[i].P_Error THEN clips[i].M_Reset('');	END_IF					
//					IF cylinders[i].P_Error THEN cylinders[i].M_Reset(''); END_IF
					
//				END_FOR
				FOR i:=0 TO 3 DO
					IF cylinders[i].xError THEN
						cylinders[i].M_Reset();
					ELSE
						cylinders[i].M_Retract();	
					END_IF
				END_FOR
					uiAbortingStep:=9000;
					
            9000:
                // Aborting process finished
				_abort:=FALSE;
                _AbortCompleted := TRUE;
        END_CASE

        IF _AbortCompleted THEN
            // Aborting process is running normally 
			uiAbortingStep:=0;
            eState := STATE_Aborted;
        ELSIF Error THEN
            // An error event occurred
            eState := STATE_ERROR;
        END_IF
END_METHOD

METHOD  M_STATE_DONE
VAR_INPUT
END_VAR
Busy := FALSE;
Done := TRUE;
RoundBeltMoveJob.HandShake.Execute:=FALSE;
RoundBeltMoveJob_Ctrl.Execute:= RoundBeltMoveJob.HandShake.Execute;

DAS_CoreSys.MachineControl.fbAllocateArea.M_ReleaseRoundBeltAccess(E_RoundBeltControlAccess.Allocating);
IF Done AND NOT Execute THEN
    eState := STATE_DORMANT;
END_IF
END_METHOD

METHOD  M_STATE_DORMANT
VAR_INPUT
END_VAR
Aborted         := FALSE;
Error           := FALSE;
ErrorID         := 0;
Busy                         := FALSE;
Done                         := FALSE;
_ResetCompleted := FALSE;
_Error          := FALSE;
_Executed       := FALSE;
_Abort			:= FALSE;
Aborted			:= FALSE;
strStatus 		:='No Error';
Status          := '';

uiExecutingStep :=uiResettingStep :=uiResumeStep :=0;
AllocationJobBatchModeReverse := E_AllocationJob.PreDataProcess;
i :=0;
j :=0;
iProcessingIndex :=0;
iWorkingCylinder :=0;
iWorkingIndex                := 0;	
Ton_RoundBeltArrivedDelay.IN := FALSE;
tAutoAllocationJobBatchTimeOut_Reverse.IN := FALSE;
bAllocateRobotMoveRequest	 := FALSE;

R1Used                       := FALSE;
R2Used                       := FALSE;
A1Used                       := FALSE;
A2Used                       := FALSE;
bMoveRotateBeltDone          := FALSE;	
bIfNextCycle				 := FALSE;	
bResettingCompleted :=FALSE;
ClipsHaveNeedle		:=
ClipsHaveNeedle_Pick:=
ClipsHaveNoNeedle	;


IF Execute THEN
	
	eSTATE:=STATE_EXECUTING;
END_IF
END_METHOD

METHOD  M_STATE_ERROR
VAR_INPUT
END_VAR
Busy                         := FALSE;
Error                        := TRUE;
tAutoAllocationJobBatchTimeOut_Reverse.IN := FALSE;
Status                       := StatusDescription;
RoundBeltMoveJob.HandShake.Execute:=FALSE;
RoundBeltMoveJob_Ctrl.Execute:= RoundBeltMoveJob.HandShake.Execute;
DAS_CoreSys.MachineControl.fbAllocateArea.M_ReleaseRoundBeltAccess(E_RoundBeltControlAccess.Allocating);
FOR i:=0 TO 3 DO
	IF cylinders[i].xError THEN
		cylinders[i].M_Reset();
	ELSE
		cylinders[i].M_Retract();	
	END_IF
END_FOR

TurnTable_Press.M_Retract();
RoundBelt_Press.M_Retract();

IF NOT Execute THEN
    eState := STATE_RESETTING;
END_IF
END_METHOD

METHOD  M_STATE_EXECUTING
VAR_INPUT
END_VAR

VAR_INST
	CurrentProcessData	: ST_AllocationJobBatchModeInfo;
	CurrentPickingCoordinates : ARRAY[0..3] OF st_Coordinate;
	CurrentPlacingCoordinates : ARRAY[0..3] OF st_Coordinate;
	CurrentSyncGroupPicking		  : ARRAY[0..3] OF UINT :=[0,1,2,3];
	CurrentSyncGroupPiacing		  : ARRAY[0..3] OF UINT :=[0,1,2,3];
	iFirstWorkIndex		:UINT;
END_VAR

VAR
	emptyCoordinate		: ST_Coordinate;
	AllocateRobot: INT;
END_VAR
		Busy := TRUE;				
			
		DAS_CoreSys.MachineControl.fbAllocateArea.M_GetRoundBeltAccess(E_RoundBeltControlAccess.Allocating);		
		RoundBeltMoveJob_Ctrl.Execute:=RoundBeltMoveJob.HandShake.Execute;
		RoundBeltMoveJob.HandShake.Busy:=RoundBeltMoveJob_Status.Busy;
		RoundBeltMoveJob.HandShake.Done:=RoundBeltMoveJob_Status.Done;
		RoundBeltMoveJob.HandShake.Error:=RoundBeltMoveJob_Status.Error;
		RoundBeltMoveJob_Position:=RoundBeltMoveJob.Position;
		
		CASE AllocationJobBatchModeReverse OF
			E_AllocationJob.PreDataProcess :
				IF NOT Pause THEN // Pausing here waiting pause finish
					
					bCheckStation:=FALSE;
					//Get current allocation data
					FOR i:=iProcessingIndex TO 	AutoAllocateJobBatch_Reverse_Ctrl.AutoMode_AllocateMoveBatch.NrOfAllocationJob-1 BY 1  DO
						CurrentProcessData := 	AutoAllocateJobBatch_Reverse_Ctrl.AutoMode_AllocateMoveBatch.AllocationInfo[iProcessingIndex];
						
						FOR j:=0 TO 3 DO
							IF NOT (CurrentProcessData.PlacingNeedleInfo[j].Station=99) THEN
									bCheckStation:=TRUE; //Station = 99 means this job should be ignou , Therefor any station of job is "not" 99 , means this job should be process
								EXIT;
							END_IF						
						END_FOR
						
						IF bCheckStation THEN
								AllocationJobBatchModeReverse:=E_AllocationJob.Idle;
								EXIT;
							ELSE
								iProcessingIndex:=iProcessingIndex+1;
								arrProcessedIndex[i] :=CurrentProcessData.ID;
						END_IF						
					END_FOR		

					IF 		AutoAllocateJobBatch_Reverse_Ctrl.AutoMode_AllocateMoveBatch.NrOfAllocationJob<= iProcessingIndex THEN
							AllocationJobBatchModeReverse:=E_AllocationJob.Finish;
					END_IF				
				END_IF
				
		
		
		
		
		
			E_AllocationJob.Idle:
				//idle 
								
				FOR i:=0 TO 3 DO
					IF CurrentProcessData.PickingNeedleInfo[i].CycleStart THEN
						FUN_GetNeedleCoordinates(uiLocation:=1,
										uiBox:=CurrentProcessData.PickingNeedleInfo[i].Box,
										uiClip:=CurrentProcessData.PickingNeedleInfo[i].Clip,
										uiNeedleLocation :=CurrentProcessData.PickingNeedleInfo[i].NeedleLocation,
										NeedleCoordinate=>CurrentPickingCoordinates[i]);
				
						CurrentSyncGroupPicking[i] :=i;
					ELSE
						CurrentPickingCoordinates[i]:=	emptyCoordinate;
						CurrentSyncGroupPicking[i] :=99;
					END_IF
					
					IF CurrentProcessData.PlacingNeedleInfo[i].CycleStart THEN
						FUN_GetNeedleCoordinates(uiLocation:=0,
										uiBox:=CurrentProcessData.PlacingNeedleInfo[i].Box,
										uiClip:=CurrentProcessData.PlacingNeedleInfo[i].Clip,
										uiNeedleLocation :=CurrentProcessData.PlacingNeedleInfo[i].NeedleLocation,
										NeedleCoordinate=>CurrentPlacingCoordinates[i]);
						CurrentSyncGroupPiacing[i] :=i;				
					ELSE
							CurrentPlacingCoordinates[i]:=	emptyCoordinate;
							CurrentSyncGroupPiacing[i] :=99;	
					END_IF
									
												
				
				
					ClipsHaveNeedle_Pick[i]:=CurrentProcessData.PickingNeedleInfo[i].CycleStart;
					ClipsHaveNeedle[i]	   :=CurrentProcessData.PlacingNeedleInfo[i].CycleStart;
					//Get placing needle info	
				END_FOR
				
				FUN_GetSyncGroup_AllocationJob(Coordinates :=CurrentPickingCoordinates,NeedleInfo:=CurrentProcessData.PickingNeedleInfo, SyncGroup=>CurrentSyncGroupPicking);
				FUN_GetSyncGroup_AllocationJob(Coordinates :=CurrentPlacingCoordinates,NeedleInfo:=CurrentProcessData.PlacingNeedleInfo, SyncGroup=>CurrentSyncGroupPiacing);	
				
				//Copy needle info to placing info
				tAutoAllocationJobBatchTimeOut_Reverse.IN:=FALSE;
				
				AllocationJobBatchModeReverse:=E_AllocationJob.Initial;
	
			E_AllocationJob.Initial:						
				//Get All cylinders & clips back
				bCheckTrue:=TRUE;
				
				tAutoAllocationJobBatchTimeOut_Reverse.IN:=TRUE	;
				
				FOR i:= 0 TO NrOfAllocateCylinder - 1 DO
					clips[i].M_Retract();//('E_AllocationJob.Initial');
					IF  clips[i].InRearPosition THEN
						cylinders[i].M_Retract();//('E_AllocationJob.Initial');			
					END_IF	
		
					IF NOT cylinders[i].InRearPosition THEN
						bCheckTrue:=FALSE;			
					END_IF
		
				END_FOR
//					IF TurnTable.Motor.Error THEN
//					TurnTable.Motor.Reset();
//					bCheckTrue:=FALSE;
//				END_IF
				
//				IF  AllocateRobot.axX.Error THEN
//					  AllocateRobot.axX.Reset();
//					  bCheckTrue:=FALSE;
//				END_IF
				
//				IF  AllocateRobot.axY.Error THEN
//					  AllocateRobot.axY.Reset();
//					  bCheckTrue:=FALSE;
//				END_IF
				
//				IF RoundBelt.Motor.Error THEN
//					RoundBelt.Motor.Reset();
//				    bCheckTrue:=FALSE;				
//				END_IF
				
				IF bCheckTrue THEN	
					tAutoAllocationJobBatchTimeOut_Reverse.IN:=FALSE	;	
					IF bAutoAllocateJobDryRun THEN
						// Dry run mode will not check if boxes is ready						
						AllocationJobBatchModeReverse:=E_AllocationJob.MoveToTargetPos;
					ELSE						
						AllocationJobBatchModeReverse:=E_AllocationJob.CheckBoxesOnTurnTableReady;
					END_IF
					
				END_IF
				IF tAutoAllocationJobBatchTimeOut_Reverse.Q THEN
					StatusDescription :='initiial Cylindes timeout';
					uiResumableStep := E_AllocationJob.Initial;
					_Abort :=TRUE;					
				END_IF
	
	E_AllocationJob.CheckBoxesOnTurnTableReady:
		//Check box is ready on turntable
		tAutoAllocationJobBatchTimeOut_Reverse.IN:=TRUE	;
		bBoxCheck :=TRUE;		
				FOR i:=0 TO 3 DO
					IF CurrentProcessdata.PickingNeedleInfo[i].CycleStart OR CurrentProcessdata.PlacingNeedleInfo[i].CycleStart THEN
						IF CurrentProcessdata.PickingNeedleInfo[i].Box=0 THEN
							R1Used :=TRUE;
							END_IF
						
						 IF  CurrentProcessdata.PickingNeedleInfo[i].Box=1 THEN
 							R2Used :=TRUE;
						END_IF
					END_IF
				END_FOR
				
				IF  R1Used THEN 
					  bBoxCheck :=INPUT.bTurnTable_I1Detect_Sensor AND bBoxCheck; 
				END_IF
				IF  R2Used THEN 
					  bBoxCheck :=INPUT.bTurnTable_I2Detect_Sensor AND bBoxCheck; 
				END_IF
 				
				IF bBoxCheck THEN
						bBoxCheck:=FALSE;
						IF NOT TurnTable_Press.InFrontPosition THEN
							TurnTable_Press.M_Extend();// .M_Extend();//('Auto Mode Allocation Batch Mode reverse : Turn table press box Forward');
						END_IF
						AllocationJobBatchModeReverse:=E_AllocationJob.MoveToTargetPos;
				END_IF
				
				IF tAutoAllocationJobBatchTimeOut_Reverse.Q THEN
					uiResumableStep := E_AllocationJob.CheckBoxesOnTurnTableReady;
					_Abort :=TRUE	;
					StatusDescription :='Box not ready on Turn table';
				END_IF
				
	E_AllocationJob.MoveToTargetPos:
				// Move to picking position
                Ton_RoundBeltArrivedDelay(IN := FALSE);
                tAutoAllocationJobBatchTimeOut_Reverse.IN := FALSE;

				IF ClipsHaveNeedle_Pick[iWorkingIndex] THEN // Work if this index is request
                	iWorkingCylinder := CurrentProcessData.PickingNeedleInfo[iWorkingIndex].Clip;
					// Get working cylinder index from picking info		
					IF cylinders[iWorkingCylinder].InRearPosition THEN
						bAllocateRobotMoveRequest	:= TRUE;			
							// Move allocating robot to picking position
						arAxisCtrl_gb[AxisNo.Allocate_X].PosMode.Acc := CurrentData.Axes.Allocate_X.HalfAuto.Acceleration;
						arAxisCtrl_gb[AxisNo.Allocate_X].PosMode.Dec := CurrentData.Axes.Allocate_X.HalfAuto.Deceleration;
						arAxisCtrl_gb[AxisNo.Allocate_X].PosMode.Jerk := CurrentData.Axes.Allocate_X.HalfAuto.Jerk;
						arAxisCtrl_gb[AxisNo.Allocate_X].PosMode.Velocity := CurrentData.Axes.Allocate_X.HalfAuto.Velocity;
						arAxisCtrl_gb[AxisNo.Allocate_X].PosMode.Position :=CurrentPickingCoordinates[iWorkingIndex].X;
					
						arAxisCtrl_gb[AxisNo.Allocate_Y].PosMode.Acc := CurrentData.Axes.Allocate_Y.HalfAuto.Acceleration;
						arAxisCtrl_gb[AxisNo.Allocate_Y].PosMode.Dec := CurrentData.Axes.Allocate_Y.HalfAuto.Deceleration;
						arAxisCtrl_gb[AxisNo.Allocate_Y].PosMode.Jerk := CurrentData.Axes.Allocate_Y.HalfAuto.Jerk;
						arAxisCtrl_gb[AxisNo.Allocate_Y].PosMode.Velocity := CurrentData.Axes.Allocate_Y.HalfAuto.Velocity;
						arAxisCtrl_gb[AxisNo.Allocate_Y].PosMode.Position := CurrentPickingCoordinates[iWorkingIndex].Y;		
					END_IF
								
              		FOR i :=0 TO 3 DO
						IF  CurrentProcessData.PlacingNeedleInfo[i].CycleStart THEN
							iFirstWorkIndex:=	i;
							EXIT;
							//Get the first working index in oreder to move the rotatebelt in Fast mode
						END_IF
					END_FOR
				

					IF CurrentProcessData.FastMode THEN //In Fast mode , RotateTable can start move at same moment 
						
		
					//	IF iCurrentRotateBeltStation <> CurrentProcessData.PlacingNeedleInfo[iFirstWorkIndex].Station THEN
							 //request to get the access to control Rotate belt
							RoundBeltMoveJob.Position:=CurrentProcessData.PlacingNeedleInfo[iFirstWorkIndex].Station;							
							RoundBeltMoveJob.HandShake.Execute		;					
							// In fast mode , just send rotatebelt to target station if it's request different station. Station check will be later
					//	END_IF
				
					END_IF
						AllocationJobBatchModeReverse:=E_AllocationJob.MovingToTargetPos;		
//    	            IF AllocateRobot.P_isMoving   THEN
						
//        	            AllocationJobBatchModeReverse := E_AllocationJob.MovingToTargetPos;					 
					
//					ELSIF	 NOT AllocateRobot.P_isMoving AND_THEN  AllocateRobot.P_InTargetPosition THEN
//						AllocationJobBatchModeReverse := E_AllocationJob.MovingToTargetPos;	
//            	    END_IF
				
				ELSE
					AllocationJobBatchModeReverse:=E_AllocationJob.IfNextPTP_Picking;	
				END_IF

     E_AllocationJob.MovingToTargetPos:

                tAutoAllocationJobBatchTimeOut_Reverse.IN := TRUE;

//                IF AllocateRobot.P_InTargetPosition THEN
//                    tAutoAllocationJobBatchTimeOut_Reverse.IN := FALSE;
//                    tAutoAllocationJobBatchTimeOut_Reverse.PT := GVL.tAutoAllocateJobCylinderTimeout;
					
//				    AllocationJobBatchModeReverse                := E_AllocationJob.CylinderDownPick;
					
//                END_IF

				IF arAxisStatus_gb[AxisNo.Allocate_X].Admin.CmdDone AND arAxisStatus_gb[AxisNo.Allocate_Y].Admin.CmdDone 
					AND arAxisStatus_gb[AxisNo.Allocate_X].Admin._OpModeAck = ModePosAbs AND arAxisStatus_gb[AxisNo.Allocate_Y].Admin._OpModeAck = ModePosAbs THEN
					bAllocateRobotMoveRequest		:= FALSE;
					AllocationJobBatchModeReverse   := E_AllocationJob.CylinderDownPick;
				END_IF
                IF tAutoAllocationJobBatchTimeOut_Reverse.Q THEN

                    StatusDescription := 'Moving to picking position timeout';
                    _Error            := TRUE;

                END_IF
				
	

            
	   E_AllocationJob.CylinderDownPick:
	   			// Cylinder move down to pick needle
                tAutoAllocationJobBatchTimeOut_Reverse.IN := TRUE;
				bCylinderCheck:=TRUE;                
                
                THIS^.cylinders[iWorkingCylinder].M_Extend();// //('AutoMode E_AllocationJob.CylinderDownPick');
				// Cylinder move down
				IF CurrentProcessData.SyncMode THEN //In sync mode , the cylinders in same sync group can move down at same step 
					FOR i := iWorkingIndex+1 TO 3 DO
						IF CurrentSyncGroupPicking[i]=CurrentSyncGroupPicking[iWorkingIndex] AND 
							ClipsHaveNeedle_Pick[i]	 THEN
							cylinders[CurrentProcessData.PickingNeedleInfo[i].Clip ].M_Extend();//('Auto Mode E_AllocationJob.CylinderDownPick in Sync placing Mode');
							bCylinderCheck :=cylinders[CurrentProcessData.PickingNeedleInfo[i].Clip ].InFrontPosition AND bCylinderCheck;			
						END_IF
					END_FOR
					
				END_IF
                
				
				
                IF cylinders[iWorkingCylinder].InFrontPosition AND bCylinderCheck THEN
                    tAutoAllocationJobBatchTimeOut_Reverse.IN := FALSE;
                    AllocationJobBatchModeReverse                := E_AllocationJob.ClipColse;
                END_IF

                IF tAutoAllocationJobBatchTimeOut_Reverse.Q THEN
					uiResumableStep := E_AllocationJob.CylinderDownPick;                    
                    _Abort            := TRUE;
					StatusDescription := 'Picking down timeout';
                END_IF

            E_AllocationJob.ClipColse:
				// Close clip to pick needke
                Ton_RoundBeltArrivedDelay.IN := FALSE;
                tAutoAllocationJobBatchTimeOut_Reverse.IN := TRUE;
				bCylinderCheck:=TRUE;
				
                THIS^.clips[iWorkingCylinder].M_Extend();//('Auto Mode E_AllocationJob.ClipColse');
						// Close clip
				IF CurrentProcessData.SyncMode THEN // In sync mode, the clips in same sync group can move together
					FOR i := iWorkingIndex+1 TO 3 DO
						IF CurrentSyncGroupPicking[i]=CurrentSyncGroupPicking[iWorkingIndex] AND 
							ClipsHaveNeedle_Pick[i]	 THEN
							clips[CurrentProcessData.PickingNeedleInfo[i].Clip ].M_Extend();//('Auto Mode E_AllocationJob.ClipColse in Sync placing Mode');
							bCylinderCheck :=clips[CurrentProcessData.PickingNeedleInfo[i].Clip ].InFrontPosition AND bCylinderCheck;			
						END_IF
					END_FOR
					
				END_IF
				
                IF clips[iWorkingCylinder].InFrontPosition AND bCylinderCheck THEN
                    tAutoAllocationJobBatchTimeOut_Reverse.IN := FALSE;
                    AllocationJobBatchModeReverse                := E_AllocationJob.CylinderUpPick;
                END_IF

                IF tAutoAllocationJobBatchTimeOut_Reverse.Q THEN

                    StatusDescription := 'Picking Close timeout';
                    uiResumableStep := E_AllocationJob.ClipColse;                    
                    _Abort            := TRUE;
                END_IF

	E_AllocationJob.CylinderUpPick:
		// Cylinder move up to pick needle
		bCylinderCheck:=TRUE;
		tAutoAllocationJobBatchTimeOut_Reverse.IN:=TRUE	;
		bBoxCheck:=TRUE;
			
		IF  R1Used THEN 
				  bBoxCheck :=INPUT.bTurnTable_I1Detect_Sensor  AND bBoxCheck; 
		END_IF
		IF  R2Used THEN 
				  bBoxCheck :=INPUT.bTurnTable_I2Detect_Sensor AND bBoxCheck; 
		END_IF
		
		THIS^.cylinders[iWorkingCylinder].M_Retract();//('Auto Mode E_AllocationJob.CylinderUpPick');		
	
		IF CurrentProcessData.SyncMode THEN
					FOR i := iWorkingIndex+1 TO 3 DO
						IF CurrentSyncGroupPicking[i]=CurrentSyncGroupPicking[iWorkingIndex] AND 
							ClipsHaveNeedle_Pick[i]	 THEN
							cylinders[CurrentProcessData.PickingNeedleInfo[i].Clip].M_Retract();//('Auto Mode E_AllocationJob.CylinderUpPick in Sync placing Mode');
							bCylinderCheck :=cylinders[CurrentProcessData.PickingNeedleInfo[i].Clip].InRearPosition AND bCylinderCheck;			
						END_IF
					END_FOR					
		END_IF
				
		IF cylinders[iWorkingCylinder].InRearPosition AND bCylinderCheck AND  bBoxCheck THEN
			R1Used:=FALSE;
			R2Used:=FALSE;
			tonFastModeTimeDelayBatch_Reverse.IN:=FALSE;		
			AllocationJobBatchModeReverse:=E_AllocationJob.IfNextPTP_Picking;
		END_IF
		
		IF tAutoAllocationJobBatchTimeOut_Reverse.Q THEN
			
			StatusDescription :='Picking Up timeout';
			uiResumableStep := E_AllocationJob.CylinderUpPick;                    
            _Abort            := TRUE;
		END_IF
		
	E_AllocationJob.IfNextPTP_Picking:
		// Check if next picking 
		iPickingNeedleCount:=1;
		IF CurrentProcessData.SyncMode THEN //Sync mode
			FOR i := iWorkingIndex+1 TO 3 DO
				IF CurrentSyncGroupPicking[i]=CurrentSyncGroupPicking[iWorkingIndex] AND 	ClipsHaveNeedle_Pick[i]	 THEN
					iPickingNeedleCount:=iPickingNeedleCount+1;
					ClipsHaveNeedle_Pick[i]:=FALSE;		
				END_IF
			END_FOR
		END_IF
		
		tAutoAllocationJobBatchTimeOut_Reverse.IN:=FALSE	;
		iWorkingIndex:=iWorkingIndex+1;
		IF iWorkingIndex>= NrOfAllocateCylinder THEN
			iWorkingIndex:=0;		
			RoundBeltMoveJob_Ctrl.Execute := FALSE;
			AllocationJobBatchModeReverse:=E_AllocationJob.CheckRotateBeltStation;	
			// If no more picking , go to next step to check  the rotate belt station 
		ELSE
			AllocationJobBatchModeReverse:=E_AllocationJob.MoveToTargetPos;
			// Still picking job , go back to next picking position
		END_IF
	
	
	E_AllocationJob.CheckRotateBeltStation:	
		// Check if the Rotate belt is in the target.
		
		IF ClipsHaveNeedle[iWorkingIndex] THEN
		
			tAutoAllocationJobBatchTimeOut_Reverse.IN:=FALSE;				
			iWorkingCylinder := CurrentProcessData.PlacingNeedleInfo[iWorkingIndex].Clip ;
			RoundBeltMoveJob.Position:=CurrentProcessData.PlacingNeedleInfo[iWorkingIndex].Station;			
			AllocationJobBatchModeReverse:=E_AllocationJob.MovingRotateBeltStation;				
		ELSE
				AllocationJobBatchModeReverse:=E_AllocationJob.IfNextPTP_Placing;	
		END_IF		
	
      E_AllocationJob.MovingRotateBeltStation:

                bMoveRotateBeltBusy := RoundBeltMoveJob_Status.Busy;
				bMoveRotateBeltDone := RoundBeltMoveJob_Status.Done;				
                RoundBeltMoveJob.HandShake.Execute := TRUE;				
				IF CurrentProcessData.FastMode THEN            
					IF cylinders[iWorkingCylinder].InRearPosition THEN
						
						bAllocateRobotMoveRequest	:= TRUE; 
                   							
						arAxisCtrl_gb[AxisNo.Allocate_X].PosMode.Acc := CurrentData.Axes.Allocate_X.HalfAuto.Acceleration;
						arAxisCtrl_gb[AxisNo.Allocate_X].PosMode.Dec := CurrentData.Axes.Allocate_X.HalfAuto.Deceleration;
						arAxisCtrl_gb[AxisNo.Allocate_X].PosMode.Jerk := CurrentData.Axes.Allocate_X.HalfAuto.Jerk;
						arAxisCtrl_gb[AxisNo.Allocate_X].PosMode.Velocity := CurrentData.Axes.Allocate_X.HalfAuto.Velocity;
						arAxisCtrl_gb[AxisNo.Allocate_X].PosMode.Position :=CurrentPlacingCoordinates[iWorkingIndex].X;
					
						arAxisCtrl_gb[AxisNo.Allocate_Y].PosMode.Acc := CurrentData.Axes.Allocate_Y.HalfAuto.Acceleration;
						arAxisCtrl_gb[AxisNo.Allocate_Y].PosMode.Dec := CurrentData.Axes.Allocate_Y.HalfAuto.Deceleration;
						arAxisCtrl_gb[AxisNo.Allocate_Y].PosMode.Jerk := CurrentData.Axes.Allocate_Y.HalfAuto.Jerk;
						arAxisCtrl_gb[AxisNo.Allocate_Y].PosMode.Velocity := CurrentData.Axes.Allocate_Y.HalfAuto.Velocity;
						arAxisCtrl_gb[AxisNo.Allocate_Y].PosMode.Position := CurrentPlacingCoordinates[iWorkingIndex].Y;		
					END_IF
                END_IF            
			
					
						
              	 IF (bMoveRotateBeltBusy OR bMoveRotateBeltDone) AND 
				    (  arAxisCtrl_gb[AxisNo.Allocate_X].Admin.Axis.Status.Moving   OR arAxisCtrl_gb[AxisNo.Allocate_Y].Admin.Axis.Status.Moving)	 THEN
					
                 	   AllocationJobBatchModeReverse := E_AllocationJob.MovedRotateBeltStation;
               	 END_IF
			
				
      E_AllocationJob.MovedRotateBeltStation:

                tAutoAllocationJobBatchTimeOut_Reverse.IN := TRUE;

                bMoveRotateBeltDone := RoundBeltMoveJob_Status.Done;
                Ton_RoundBeltArrivedDelay(IN := bMoveRotateBeltDone);

                IF bMoveRotateBeltDone THEN
					RoundBeltMoveJob.HandShake.Execute := FALSE;  
					IF CurrentProcessData.FastMode THEN   
                   	     AllocationJobBatchModeReverse   :=E_AllocationJob.MovingToPlacingPos;          	 
					 
					 ELSE
					 	AllocationJobBatchModeReverse := E_AllocationJob.MoveToPlacingPos; 					 
					 END_IF
                END_IF
				
			 

                IF tAutoAllocationJobBatchTimeOut_Reverse.Q THEN

                    StatusDescription := 'Rotate Belt TimeOut';
                    _Error            := TRUE;

                END_IF
	
            E_AllocationJob.MoveToPlacingPos:

                IF ClipsHaveNeedle[iWorkingIndex] THEN 
                    iWorkingCylinder := CurrentProcessData.PlacingNeedleInfo[iWorkingIndex].Clip;
					IF cylinders[iWorkingCylinder].InRearPosition THEN
						
						bAllocateRobotMoveRequest	:= TRUE;
                  
						arAxisCtrl_gb[AxisNo.Allocate_X].PosMode.Acc := CurrentData.Axes.Allocate_X.HalfAuto.Acceleration;
						arAxisCtrl_gb[AxisNo.Allocate_X].PosMode.Dec := CurrentData.Axes.Allocate_X.HalfAuto.Deceleration;
						arAxisCtrl_gb[AxisNo.Allocate_X].PosMode.Jerk := CurrentData.Axes.Allocate_X.HalfAuto.Jerk;
						arAxisCtrl_gb[AxisNo.Allocate_X].PosMode.Velocity := CurrentData.Axes.Allocate_X.HalfAuto.Velocity;
						arAxisCtrl_gb[AxisNo.Allocate_X].PosMode.Position :=CurrentPlacingCoordinates[iWorkingIndex].X;
					
						arAxisCtrl_gb[AxisNo.Allocate_Y].PosMode.Acc := CurrentData.Axes.Allocate_Y.HalfAuto.Acceleration;
						arAxisCtrl_gb[AxisNo.Allocate_Y].PosMode.Dec := CurrentData.Axes.Allocate_Y.HalfAuto.Deceleration;
						arAxisCtrl_gb[AxisNo.Allocate_Y].PosMode.Jerk := CurrentData.Axes.Allocate_Y.HalfAuto.Jerk;
						arAxisCtrl_gb[AxisNo.Allocate_Y].PosMode.Velocity := CurrentData.Axes.Allocate_Y.HalfAuto.Velocity;
						arAxisCtrl_gb[AxisNo.Allocate_Y].PosMode.Position := CurrentPlacingCoordinates[iWorkingIndex].Y;		
							
                        AllocationJobBatchModeReverse := E_AllocationJob.MovingToPlacingPos;         
					END_IF           

                ELSE

                    AllocationJobBatchModeReverse := E_AllocationJob.IfNextPTP_Placing;
                END_IF
				
	

            E_AllocationJob.MovingToPlacingPos:

                tAutoAllocationJobBatchTimeOut_Reverse.IN := TRUE;           		 
				IF arAxisStatus_gb[AxisNo.Allocate_X].Admin.CmdDone 
					AND arAxisStatus_gb[AxisNo.Allocate_Y].Admin.CmdDone
					AND arAxisStatus_gb[AxisNo.Allocate_X].Admin._OpModeAck = ModePosAbs
					AND arAxisStatus_gb[AxisNo.Allocate_Y].Admin._OpModeAck = ModePosAbs
					AND NOT arAxisCtrl_gb[AxisNo.RoundBelt].Admin.Axis.Status.Moving 
					AND  arAxisCtrl_gb[AxisNo.Allocate_X].Admin.Axis.Status.NotMoving
					AND  arAxisCtrl_gb[AxisNo.Allocate_Y].Admin.Axis.Status.NotMoving		THEN
					bAllocateRobotMoveRequest := FALSE;
					RoundBeltMoveJob.HandShake.Execute := FALSE; 
					tAutoAllocationJobBatchTimeOut_Reverse.IN := FALSE;
					IF RoundBelt_Press.InFrontPosition THEN // make sure press box cylinder is in front
							IF bAutoAllocateJobDryRun THEN
	                 		   AllocationJobBatchModeReverse                := E_AllocationJob.CylinderDownPlace;
							ELSE
								AllocationJobBatchModeReverse                := E_AllocationJob.CheckBoxReadyOnAllocatePosOfRoundBelt;
							END_IF
						ELSE
							RoundBelt_Press.M_Extend();//('');	
						END_IF
					
				END_IF
               

                IF tAutoAllocationJobBatchTimeOut_Reverse.Q THEN

                    StatusDescription := 'Moving placing timeout';
                    _Error            := TRUE;

                END_IF

			E_AllocationJob.CheckBoxReadyOnAllocatePosOfRoundBelt:
				tAutoAllocationJobBatchTimeOut_Reverse.IN:=TRUE	;				
				
				  FOR i:=0 TO 3 DO
					IF CurrentProcessData.PlacingNeedleInfo[iWorkingIndex].Station = CurrentProcessData.PlacingNeedleInfo[i].Station THEN
						IF CurrentProcessData.PlacingNeedleInfo[i].Box=0 THEN
							A1Used :=TRUE;
							END_IF
						
					 	IF  CurrentProcessData.PlacingNeedleInfo[i].Box=1 THEN
 							A2Used :=TRUE;
						END_IF
					END_IF
				  END_FOR
				
				  IF  A1Used THEN 
					  bBoxCheck :=INPUT.bRoundBelt_WorkZoneQ1Detect_Sensor AND bBoxCheck; 
				  END_IF
				  IF  A2Used THEN 
					  bBoxCheck :=INPUT.bRoundBelt_WorkZoneQ2Detect_Sensor AND bBoxCheck; 
				  END_IF
 				
				  IF bBoxCheck THEN
						AllocationJobBatchModeReverse:=E_AllocationJob.CylinderDownPlace;
						A1Used := A2Used := FALSE;
				  END_IF
				
				IF tAutoAllocationJobBatchTimeOut_Reverse.Q THEN
					_Error :=TRUE	;
					StatusDescription :='Box not ready on Rotate Belt';
				END_IF	
				
            E_AllocationJob.CylinderDownPlace:
                bCylinderCheck               := TRUE;
                tAutoAllocationJobBatchTimeOut_Reverse.IN := TRUE;
                cylinders[iWorkingCylinder].M_Extend();//('Auto Mode E_AllocationJob.CylinderDownPlace');
				
				IF CurrentProcessData.SyncMode THEN
					FOR i := iWorkingIndex+1 TO 3 DO
						IF CurrentSyncGroupPiacing[i]=CurrentSyncGroupPiacing[iWorkingIndex] AND 
							ClipsHaveNeedle[i]	 THEN
							cylinders[CurrentProcessData.PlacingNeedleInfo[i].Clip].M_Extend();//('Auto Mode E_AllocationJob.CylinderDownPlace in Sync placing Mode');
							//bCylinderCheck :=cylinders[i].InFrontPosition AND bCylinderCheck;		
							bCylinderCheck :=cylinders[CurrentProcessData.PlacingNeedleInfo[i].Clip].InFrontPosition AND bCylinderCheck;
						END_IF
					END_FOR
					
				END_IF
				
               	 IF cylinders[iWorkingCylinder].InFrontPosition AND bCylinderCheck THEN
                    tAutoAllocationJobBatchTimeOut_Reverse.IN := FALSE;
                    AllocationJobBatchModeReverse                := E_AllocationJob.ClipOpen;
              	  END_IF
				
                IF tAutoAllocationJobBatchTimeOut_Reverse.Q THEN
                    StatusDescription := ' placing down timeout';
                    uiResumableStep := E_AllocationJob.CylinderDownPlace;                    
           			 _Abort            := TRUE;
                END_IF

            E_AllocationJob.ClipOpen:
                tAutoAllocationJobBatchTimeOut_Reverse.IN := TRUE;
                bCylinderCheck               := TRUE;
                clips[iWorkingCylinder].M_Retract();//('Auto Mode E_AllocationJob.ClipOpen');
					IF CurrentProcessData.SyncMode THEN
					FOR i := iWorkingIndex+1 TO 3 DO
						IF CurrentSyncGroupPiacing[i]=CurrentSyncGroupPiacing[iWorkingIndex] AND 
							ClipsHaveNeedle[i]	 THEN
							clips[CurrentProcessData.PlacingNeedleInfo[i].Clip].M_Retract();//('Auto Mode E_AllocationJob.ClipOpen in Sync placing Mode');
//							bCylinderCheck :=clips[i].InRearPosition AND bCylinderCheck;		
							bCylinderCheck :=clips[CurrentProcessData.PlacingNeedleInfo[i].Clip].InRearPosition AND bCylinderCheck;	
						END_IF
					END_FOR
					
				END_IF
				
				
                IF clips[iWorkingCylinder].InRearPosition AND bCylinderCheck THEN
                    tAutoAllocationJobBatchTimeOut_Reverse.IN := FALSE;
                    AllocationJobBatchModeReverse                := E_AllocationJob.CylinderUpPlace;
                END_IF

                IF tAutoAllocationJobBatchTimeOut_Reverse.Q THEN

                    StatusDescription := ' placing Close timeout';
                    uiResumableStep := E_AllocationJob.ClipOpen;                    
           			 _Abort            := TRUE;
                END_IF

            E_AllocationJob.CylinderUpPlace:
                bCylinderCheck         := TRUE;
                //bCylinderCheckFastMode := TRUE;

                cylinders[iWorkingCylinder].M_Retract();//(' Auto Mode E_AllocationJob.CylinderUpPlace');
				
					IF CurrentProcessData.SyncMode THEN
					FOR i := iWorkingIndex+1 TO 3 DO
						IF CurrentSyncGroupPiacing[i]=CurrentSyncGroupPiacing[iWorkingIndex] AND 
							ClipsHaveNeedle[i]	 THEN
							cylinders[CurrentProcessData.PlacingNeedleInfo[i].Clip].M_Retract();//('Auto Mode E_AllocationJob.CylinderUpPlace in Sync placing Mode');
							bCylinderCheck :=cylinders[CurrentProcessData.PlacingNeedleInfo[i].Clip].InRearPosition AND bCylinderCheck;	
							//bCylinderCheckFastMode := (NOT cylinders[i].InRearPosition) AND bCylinderCheckFastMode;
							
						END_IF
					END_FOR					
				END_IF
(*==========================	取消FastMode，預防偷跑導致機構衝突。//edited by Gamin，2026/03/31
				IF CurrentProcessData.FastMode  AND NOT cylinders[iWorkingCylinder].InFrontPosition AND bCylinderCheckFastMode THEN						
               		 tonFastModeTimeDelayBatch_Reverse.IN := TRUE;
				END_IF
				
                IF (cylinders[iWorkingCylinder].InRearPosition AND bCylinderCheck) OR  tonFastModeTimeDelayBatch_Reverse.Q THEN
                    tAutoAllocationJobBatchTimeOut_Reverse.IN              := FALSE;
					tonFastModeTimeDelayBatch_Reverse.IN 				  := FALSE;
                   // GVL.TwinCatMemory.AllocatingInfoToHost[1] := THIS^.AutoAllocateJob_Ctrl.AutoMode_AllocateMove.PlacingNeedleInfo[iWorkingIndex];
                    //Update TwinCat memory
                    AllocationJobBatchModeReverse := E_AllocationJob.CheckNeedlePlaced;

                END_IF
=============================*)
				 IF cylinders[iWorkingCylinder].InRearPosition AND bCylinderCheck THEN
                    tAutoAllocationJobBatchTimeOut_Reverse.IN              := FALSE;
                    AllocationJobBatchModeReverse := E_AllocationJob.CheckNeedlePlaced;
                END_IF

                IF tAutoAllocationJobBatchTimeOut_Reverse.Q THEN
                    StatusDescription := ' placing Up timeout';
                    uiResumableStep := E_AllocationJob.CylinderUpPlace;                    
           			 _Abort            := TRUE;
                END_IF

			E_AllocationJob.CheckNeedlePlaced: 
				ClipsHaveNeedle[iWorkingIndex] :=FALSE;
				IF CurrentProcessData.SyncMode THEN
					FOR i := iWorkingIndex+1 TO 3 DO
						IF CurrentSyncGroupPiacing[i]=CurrentSyncGroupPiacing[iWorkingIndex] AND ClipsHaveNeedle[i]	 THEN
							ClipsHaveNeedle[i]:=FALSE;
						END_IF
					END_FOR		
				END_IF
				AllocationJobBatchModeReverse := E_AllocationJob.IfNextPTP_Placing;
				
            E_AllocationJob.IfNextPTP_Placing:
                iWorkingIndex := iWorkingIndex + 1;

                IF iWorkingIndex >= NrOfAllocateCylinder THEN
                    iWorkingIndex := 0;
                    AllocationJobBatchModeReverse := E_AllocationJob.Finish;
                ELSE

                    AllocationJobBatchModeReverse := E_AllocationJob.CheckRotateBeltStation;
                END_IF

           
            E_AllocationJob.Finish:
                // Finish

               	arrProcessedIndex[iProcessingIndex] :=CurrentProcessData.ID;					
				IF 	AutoAllocateJobBatch_Reverse_Ctrl.AutoMode_AllocateMoveBatch.NrOfAllocationJob> iProcessingIndex+1 THEN			
					
					iProcessingIndex :=iProcessingIndex+1;
					AllocationJobBatchModeReverse := E_AllocationJob.PreDataProcess;
				ELSE
					_Executed := TRUE;
				END_IF				
        END_CASE	
			


	

IF NOT Execute THEN
	eState:=STATE_RESETTING;
END_IF
IF _Error THEN
	eState:=STATE_ERROR;
END_IF
IF _Abort THEN
	eSTATE:=STATE_ABORTING;
END_IF
IF _Executed THEN
	eSTATE:=STATE_Done;
END_IF
END_METHOD

METHOD  M_STATE_RESETTING
VAR_INPUT
END_VAR
Busy                         := FALSE;
Done                         := FALSE;
Error                        := FALSE;
_Error                       := FALSE;
tAutoAllocationJobBatchTimeOut_Reverse.IN := FALSE;

  CASE uiResettingStep OF
            0:
                // Resetting process start

                uiAbortingStep := 0;
                uiAbortedStep  := 0;
				RoundBeltMoveJob_Ctrl.Execute:=FALSE;
                IF M_CheckClipsNoError() AND_THEN
                   M_CheckCylindersNoError()
                THEN
                    // no error -> no need to reset
                    bResettingCompleted := TRUE;
                ELSE
                    uiResettingStep := 1000;
                END_IF

            1000:

//                FOR i := 1 TO GVL.NrOfAllocateCylinder DO
//                    IF THIS^.Clips[i].bError THEN
//                        THIS^.Clips[i].M_Reset('Auto Allocating Job Reset');
//                    END_IF

//                    IF THIS^.cylinders[i].bError THEN
//                        THIS^.cylinders[i].M_Reset('Auto Allocating Job Reset');
//                    END_IF
//                END_FOR
				DAS_CoreSys.MachineControl.fbAllocateArea.M_ReleaseRoundBeltAccess(E_RoundBeltControlAccess.Allocating);
                uiResettingStep := 2000;
			
			2000:
//					IF TurnTable.Motor.Error THEN
//					TurnTable.Motor.Reset();
//				END_IF
				
//				IF  AllocateRobot.axX.Error THEN
//					  AllocateRobot.axX.Reset();
//				END_IF
				
//				IF  AllocateRobot.axY.Error THEN
//					  AllocateRobot.axY.Reset();
//				END_IF
				
//				IF RoundBelt.Motor.Error THEN
//					RoundBelt.Motor.Reset();			
//				END_IF
				uiResettingStep := 9000;
				
            9000:
                // Resetting process is finished
                bResettingCompleted := TRUE;
        END_CASE

        IF bResettingCompleted THEN
            eState := STATE_DORMANT;
        END_IF
END_METHOD

END_FUNCTION_BLOCK

// ---- Library/20_MachineUnits/22_AllocateArea/Old_Version_Service/FB_OutRobot_BoxMoveReverse_Old.TcPOU
FUNCTION_BLOCK FB_OutRobot_BoxMoveReverse_Old EXTENDS FB_ObjectBase_V2
VAR_INPUT
//    Execute    :BOOL;   // True : This prog will start.
//    Abort      :BOOL;   // True : This prog will be abort.
//    Reset      :BOOL;   // True : This prog will be reset.
//    ObjectName :STRING; // Set this fb name(About it's action)
	INPUT            			   : REFERENCE TO ST_InputTable;
	Cylinder   					   : REFERENCE TO UNI_CylinderList;
	Motor      					   : REFERENCE TO UNI_MotorList;
	Cylinders					   : REFERENCE TO ARRAY[0..1] OF FB_Cylinder;
	Clips						   : REFERENCE TO ARRAY[0..1] OF FB_Cylinder;
	AutoMode_OutRobotMoveMove : st_AutoMode_ClampingBoxesJob;	
END_VAR

VAR_OUTPUT
//    Busy    :BOOL;        // True : This prog is running.
//    Done    :BOOL;        // True : Command has been executed.
//    Aborted :BOOL;        // True : This prog is aborted.
//    Error   :BOOL;        // True : This prog has an error.
//    ErrorID :UINT;       // Output ErrorID
//    Status  :T_MaxString; // Output this prog status by string(255bytes)
END_VAR

VAR
//    eState :E_MethodStatus_Basic;
//	uiExecutingStep : UDINT; // This var is used to been controll STATE_EXECUTING process.
//	uiResettingStep : UDINT;
//	uiAbortingStep : UDINT;
//	_Executed :BOOL; // Executing process completed.
//	_Error : BOOL; // FB has an error.
//	_ResetCompleted : BOOL; // FB resetting completed.
//	_AbortCompleted : BOOL; // FB aborting completed.
	//_Abort		: BOOL;
	strStatus	: STRING;
	uiResumeStep : UINT;
	tonTimeOut   :TON;
	tonTimeDelay   :TON;
	iWorkingIndex : INT;
	_UniqueErrorCode :STRING;
	
	
	PickingPos	: ARRAY[0..1] OF ST_PositionTable;
	PlacingPos  : ARRAY[0..1] OF ST_PositionTable;
	bSyncPick	: BOOL;
	bSyncPlace	: BOOL;
	SensorOnConveyor			   : BIT;
	ConveyorMotor				   : REFERENCE TO FB_Motor;
	UseA	: BOOL;
	UseB	: BOOL;
	bMotorMoveForward : BOOL;
END_VAR

A00_BasicUnits();
SUPER^.A10_StateControl();

ACTION A00_BasicUnits:
tonTimeOut(PT:=T#60S);
tonTimeDelay(PT:=T#1.5s);
END_ACTION

METHOD GetModelState
VAR_OUTPUT
    xDone    :BOOL;
    xBusy    :BOOL;
    xError   :BOOL;
    xAborted :BOOL;
    iErrorID :UDINT;
	UniqueErrorCode : STRING;
END_VAR
xDone    := Done;
xBusy    := Busy;
xError   := Error;
xAborted := Abort;
iErrorID := ErrorID;
UniqueErrorCode := THIS^.UniqueErrorCode;
END_METHOD

METHOD GetName : STRING
GetName := ObjectName;
END_METHOD

METHOD PRIVATE M_CheckCommand : BOOL
VAR_INPUT
END_VAR


M_CheckCommand:=true;
END_METHOD

METHOD PRIVATE M_GetWorkingConditions : BOOL
VAR_INPUT
END_VAR
//For Outbox move reverse, Boxes must place on same position , therefor only work with TargetPosition of ClipA

IF AutoMode_OutRobotMoveMove.ClampingInfo.TargetOfClipA = 5 THEN
	ConveyorMotor REF= Motor.List.TransmitDifferentSideCV;
ELSIF AutoMode_OutRobotMoveMove.ClampingInfo.TargetOfClipA = 6 THEN
	ConveyorMotor REF= Motor.List.TransmitSameSideCV;
ELSIF AutoMode_OutRobotMoveMove.ClampingInfo.TargetOfClipA = 3 THEN
	ConveyorMotor REF= Motor.List.TransmitDifferentSideCV;
ELSIF AutoMode_OutRobotMoveMove.ClampingInfo.TargetOfClipA = 4 THEN
	ConveyorMotor REF= Motor.List.TransmitSameSideCV;	
END_IF

IF AutoMode_OutRobotMoveMove.ClampingInfo.TargetOfClipA=5 THEN
		bMotorMoveForward := FALSE;
	ELSE
		bMotorMoveForward := TRUE;	
END_IF
IF AutoMode_OutRobotMoveMove.ClampingInfo.UseClibA THEN
	PickingPos[0] :=FUN_GetPositionTableData('R',1,0);
	UseA := TRUE;
	CASE  AutoMode_OutRobotMoveMove.ClampingInfo.TargetOfClipA OF	
		
	3,4:
		PlacingPos[0] :=FUN_GetPositionTableData('O',AutoMode_OutRobotMoveMove.ClampingInfo.TargetOfClipA,0);
	5,6:
		PlacingPos[0] :=FUN_GetPositionTableData('I',AutoMode_OutRobotMoveMove.ClampingInfo.TargetOfClipA,0);
	ELSE
		strStatus :='FB_OutRobot_BoxMoveReverse: Wrong command: Clip A target not allow';
		M_GetWorkingConditions := FALSE;
		RETURN;
	END_CASE
END_IF

IF AutoMode_OutRobotMoveMove.ClampingInfo.UseClibB THEN
	PickingPos[1] :=FUN_GetPositionTableData('R',2,1);
	UseB :=TRUE;
		CASE AutoMode_OutRobotMoveMove.ClampingInfo.TargetOfClipA OF
		
	3,4:
		PlacingPos[1] :=FUN_GetPositionTableData('O',AutoMode_OutRobotMoveMove.ClampingInfo.TargetOfClipA,1);
	5,6 :
		PlacingPos[1] :=FUN_GetPositionTableData('I',AutoMode_OutRobotMoveMove.ClampingInfo.TargetOfClipA,1);
	ELSE
		strStatus :='FB_OutRobot_BoxMoveReverse: Wrong command: Clip B target not allow';
		M_GetWorkingConditions := FALSE;
		RETURN;
	END_CASE
END_IF
IF PlacingPos[0].X_Pos =PlacingPos[1].X_Pos AND PlacingPos[0].Y_Pos = PlacingPos[1].Y_Pos AND UseA AND UseB THEN
		bSyncPlace:=TRUE;
	ELSE
		bSyncPlace:=FALSE;	
END_IF
IF PickingPos[0].X_Pos =PickingPos[1].X_Pos AND PickingPos[0].Y_Pos = PickingPos[1].Y_Pos AND UseA AND UseB THEN
		bSyncPick:=TRUE;
	ELSE
		bSyncPick:=FALSE;	
END_IF

M_GetWorkingConditions :=TRUE;
END_METHOD

METHOD PRIVATE M_RecoveryAllObjects : BOOL
VAR_INPUT
END_VAR
VAR 
	i : INT;
END_VAR
FOR i:=0 TO 1 DO
	IF Clips[i].xError THEN
		Clips[i].M_Reset();
		ELSE
		Clips[i].M_Retract();		
	END_IF
	IF Cylinders[i].xError THEN
	Cylinders[i].M_Reset();	
	ELSE
	Cylinders[i].M_Retract();	
	END_IF
END_FOR


IF arAxisCtrl_gb[AxisNo.OutRobot_X].Admin.Axis.Status.Error THEN

	arAxisCtrl_gb[AxisNo.OutRobot_X].Admin.ClearError:= TRUE;
ELSE
	arAxisCtrl_gb[AxisNo.OutRobot_X].Admin.ClearError:= FALSE;
END_IF

IF arAxisCtrl_gb[AxisNo.OutRobot_Y].Admin.Axis.Status.Error THEN

	arAxisCtrl_gb[AxisNo.OutRobot_Y].Admin.ClearError:= TRUE;
ELSE
	arAxisCtrl_gb[AxisNo.OutRobot_Y].Admin.ClearError:= FALSE;
END_IF
END_METHOD

METHOD PRIVATE M_SensorUpdate : BOOL
VAR_INPUT
END_VAR
IF AutoMode_OutRobotMoveMove.ClampingInfo.TargetOfClipA = 5 THEN
	SensorOnConveyor := INPUT.bDifferentSizeCV_BoxDetect5_Sensor;
ELSIF AutoMode_OutRobotMoveMove.ClampingInfo.TargetOfClipA = 6 THEN
	SensorOnConveyor := INPUT.bSameSizeCV_BoxDetect5_Sensor;
ELSIF AutoMode_OutRobotMoveMove.ClampingInfo.TargetOfClipA = 3 THEN
	SensorOnConveyor := INPUT.bDifferentSizeCV_BoxDetect4_Sensor;
ELSIF AutoMode_OutRobotMoveMove.ClampingInfo.TargetOfClipA = 4 THEN
	SensorOnConveyor := INPUT.bSameSizeCV_BoxDetect4_Sensor;	
END_IF
END_METHOD

METHOD  M_STATE_ABORTED
VAR_INPUT
END_VAR
ERROR :=TRUE;
Busy    := FALSE;
Aborted := TRUE;
Status := strStatus;

IF NOT Execute THEN
	eSTATE:=STATE_RESETTING;
END_IF

IF Execute AND Reset THEN
//	uiExecutingStep :=uiResumeStep;
	eSTATE:=STATE_EXECUTING;
END_IF
END_METHOD

METHOD  M_STATE_ABORTING
VAR_INPUT
END_VAR

VAR
	i : int;
	bCylinderCheck: BOOL;
END_VAR
Error :=True;
CASE uiAbortingStep OF
	0 :
		bCylinderCheck:=TRUE;
		ConveyorMotor.M_MotorStop();
		FOR i :=0 TO 1 DO		
	    	Cylinders[i].M_Reset();
			Cylinders[i].M_Retract();
			bCylinderCheck:=bCylinderCheck AND Cylinders[i].InRearPosition;	
		END_FOR
		IF bCylinderCheck THEN		
			uiAbortingStep:=9999;
		END_IF
		
	9999:	
			_AbortCompleted:=TRUE;
END_CASE

IF _AbortCompleted THEN	
	eSTATE :=STATE_ABORTED;
END_IF
END_METHOD

METHOD  M_STATE_DONE
VAR_INPUT
END_VAR
Busy 	:= FALSE;
Done	:=TRUE;

IF NOT Execute THEN
	eSTATE:=STATE_RESETTING;
END_IF
END_METHOD

METHOD  M_STATE_DORMANT
VAR_INPUT
END_VAR
Busy            := FALSE;
Done            := FALSE;
Aborted         := FALSE;
Error           := FALSE;
ErrorID         := 0;
Status          := '';
_ResetCompleted := FALSE;
_Error          := FALSE;
_Executed       := FALSE;
strStatus :='FB_OutRobot_BoxMoveReverse: No Error';
uiExecutingStep :=uiResettingStep :=uiResumeStep :=0;
tonTimeOut.IN :=TRUE;
_UniqueErrorCode:='0';
iWorkingIndex :=0;
bSyncPick :=FALSE;
bSyncPlace := FALSE;
UseA := FALSE;
UseB :=FALSE;
bMotorMoveForward:= FALSE;

IF Execute THEN
	eSTATE:=STATE_EXECUTING;
END_IF
END_METHOD

METHOD  M_STATE_ERROR
VAR_INPUT
END_VAR
ERROR   :=TRUE;
Busy	:=FALSE;
Status := strStatus;
ConveyorMotor.M_MotorStop();

IF NOT Execute THEN	
eSTATE:=STATE_RESETTING;
END_IF
END_METHOD

METHOD  M_STATE_EXECUTING
VAR_INPUT
END_VAR
VAR_INST
	bMoveConveyorForward : BOOL;
	bMoveConveyorBackrward : bool;
END_VAR

VAR
	bCylinderCheck : BOOL := TRUE;
END_VAR
Busy :=TRUE;
M_SensorUpdate();
IF bMoveConveyorForward THEN
	IF NOT ConveyorMotor.InBackWard THEN
		ConveyorMotor.M_MoveForward();	
	END_IF
END_IF

IF bMoveConveyorBackrward THEN
	IF NOT ConveyorMotor.InForWard THEN
		ConveyorMotor.M_MoveBackward();
	END_IF
END_IF
CASE uiExecutingStep OF
	

0: //Idle
bMoveConveyorForward:=FALSE;
bMoveConveyorBackrward:=FALSE;
	tonTimeDelay.IN :=FALSE;
	tonTimeOut.IN := FALSE;
	M_RecoveryAllObjects();
	//M_GetWorkingConditions();
	iWorkingIndex :=0;
	uiExecutingStep := 100;
	
100: //Check command
	IF M_GetWorkingConditions()THEN
		uiExecutingStep:=200;
	ELSE
		_Error:=TRUE;		
	END_IF
	
200: // first index

		IF UseA THEN
			iWorkingIndex :=0;
		ELSE
			iWorkingIndex :=1;	
		END_IF
		
		uiExecutingStep:=1000;	
	
1000: 
	// Move OutRobot to First clip picking	
	 	 
	arAxisCtrl_gb[AxisNo.OutRobot_X].PosMode.Position := PickingPos[iWorkingIndex].X_Pos;		
	arAxisCtrl_gb[AxisNo.OutRobot_Y].PosMode.Position := PickingPos[iWorkingIndex].Y_Pos;	
	uiExecutingStep:=1100;
		// todo : Check axes is moving
1100:
	// Check outRobot arrived
	IF		(arAxisStatus_gb[AxisNo.OutRobot_X].Admin._OpModeAck = ModePosAbs AND arAxisStatus_gb[AxisNo.OutRobot_X].Admin.CmdDone) 
	AND (arAxisStatus_gb[AxisNo.OutRobot_Y].Admin._OpModeAck = ModePosAbs AND arAxisStatus_gb[AxisNo.OutRobot_Y].Admin.CmdDone) 
	THEN
		tonTimeOut.IN := FALSE;
		uiExecutingStep:=1200;
	END_IF	
	tonTimeOut.IN := TRUE;
	IF tonTimeOut.q THEN
		tonTimeOut.IN := FALSE;
		_Error := TRUE;
		strStatus :='FB_OutRobot_BoxMoveReverse Step 1100: Move Robot to picking position timeout';
	END_IF
1200: //Clip Down Pick	  
	bCylinderCheck := TRUE;
	Cylinders[iWorkingIndex].M_Extend();
	bCylinderCheck := Cylinders[iWorkingIndex].InFrontPosition AND bCylinderCheck;
	IF bSyncPick THEN
		Cylinders[1].M_Extend();
		bCylinderCheck := Cylinders[1].InFrontPosition AND bCylinderCheck;
	END_IF	
	 
	IF bCylinderCheck THEN
		tonTimeOut.IN := FALSE;
		uiExecutingStep:=1300;
	END_IF 
	tonTimeOut.IN := TRUE;
	IF tonTimeOut.q THEN
		tonTimeOut.IN := FALSE;
		_Abort := TRUE;
		strStatus :='FB_OutRobot_BoxMoveReverse Step 1200: Cylinder pick down timeout';
	END_IF
	
1300: // Clip close Pick
	bCylinderCheck := TRUE;
	Clips[iWorkingIndex].M_Extend();
	bCylinderCheck := Clips[iWorkingIndex].InFrontPosition AND bCylinderCheck;
	IF bSyncPick THEN
		Clips[1].M_Extend();
		bCylinderCheck := Clips[1].InFrontPosition AND bCylinderCheck;
	END_IF	
	 
	IF bCylinderCheck THEN
		tonTimeOut.IN := FALSE;
		uiExecutingStep:=1400;
	END_IF 
	tonTimeOut.IN := TRUE;
	IF tonTimeOut.q THEN
		tonTimeOut.IN := FALSE;
		_Abort := TRUE;
		strStatus :='FB_OutRobot_BoxMoveReverse Step 1300: Clip pick close timeout';
	END_IF
	
1400: // Clip Up Pick
	bCylinderCheck := TRUE;
	Cylinders[iWorkingIndex].M_Retract();
	bCylinderCheck := Cylinders[iWorkingIndex].InRearPosition AND bCylinderCheck;
	IF bSyncPick THEN
		Cylinders[1].M_Retract();
		bCylinderCheck := Cylinders[1].InRearPosition AND bCylinderCheck;
	END_IF	
	 
	IF bCylinderCheck THEN
		tonTimeOut.IN := FALSE;
		uiExecutingStep:=1500;
	END_IF 
	  tonTimeOut.IN := TRUE;
	IF tonTimeOut.q THEN
		tonTimeOut.IN := FALSE;
		_Abort := TRUE;
		strStatus :='FB_OutRobot_BoxMoveReverse Step 1400: Cylinder pick up timeout';
	END_IF
	
1500: // If Next pick
	  IF iWorkingIndex>=1 OR bSyncPick OR NOT UseB THEN
		//Go to placing step
			IF UseA THEN
				iWorkingIndex:=0;
			ELSE
				iWorkingIndex:=1;	
			END_IF
			uiExecutingStep:=2000;
		ELSE
			iWorkingIndex :=iWorkingIndex +1;
			uiExecutingStep:=1000;	
	  END_IF
	  

2000: // Move to Placing pos
	  // Move Conveyor 
	   IF bMotorMoveForward THEN
		 	bMoveConveyorForward:=TRUE;//ConveyorMotor.M_MoveForward();
			bMoveConveyorBackrward := FALSE;
		  ELSE	 
			  bMoveConveyorForward := FALSE;
			 bMoveConveyorBackrward := TRUE; 
	 		 ConveyorMotor.M_MoveBackward(); 
	   END_IF
	   
	 arAxisCtrl_gb[AxisNo.OutRobot_X].PosMode.Position := PlacingPos[iWorkingIndex].X_Pos;		
	 arAxisCtrl_gb[AxisNo.OutRobot_Y].PosMode.Position := PlacingPos[iWorkingIndex].Y_Pos;	
	 uiExecutingStep:=2100;

2100: // Waiting outRobot move to placing pos	 
	  // Check sensor off for a while
	tonTimeDelay.IN := NOT 	SensorOnConveyor;
	 IF	(arAxisStatus_gb[AxisNo.OutRobot_X].Admin._OpModeAck = ModePosAbs AND arAxisStatus_gb[AxisNo.OutRobot_X].Admin.CmdDone) 
	AND (arAxisStatus_gb[AxisNo.OutRobot_Y].Admin._OpModeAck = ModePosAbs AND arAxisStatus_gb[AxisNo.OutRobot_Y].Admin.CmdDone)
	AND  tonTimeDelay.Q
	THEN	
		tonTimeOut.IN := FALSE;	
		uiExecutingStep:=2150;
	END_IF	
	
	  tonTimeOut.IN := TRUE;
	IF tonTimeOut.q THEN
		tonTimeOut.IN := FALSE;
		_Error := TRUE;
		strStatus :='FB_OutRobot_BoxMoveReverse Step 2100: Move Robot to placing position time out';
	END_IF
	
2150 : //Motor stop
		tonTimeDelay.IN := FALSE;
		bMoveConveyorForward:=FALSE;
		bMoveConveyorBackrward:=FALSE;
		ConveyorMotor.M_MotorStop();
		IF	ConveyorMotor.InStopped THEN
			uiExecutingStep:=2200;
		END_IF

2200: //Cllp Down place
	bCylinderCheck := TRUE;
	Cylinders[iWorkingIndex].M_Extend();
	bCylinderCheck := Cylinders[iWorkingIndex].InFrontPosition AND bCylinderCheck;
	IF bSyncPlace THEN
		Cylinders[1].M_Extend();
		bCylinderCheck := Cylinders[1].InFrontPosition AND bCylinderCheck;
	END_IF	
	 
	IF bCylinderCheck THEN
		tonTimeOut.IN := FALSE;
		uiExecutingStep:=2300;
	END_IF 
	
	  tonTimeOut.IN := TRUE;
	IF tonTimeOut.q THEN
		tonTimeOut.IN := FALSE;
		_Abort := TRUE;
		strStatus :='FB_OutRobot_BoxMoveReverse Step 2200: Cylinder place down timeout';
	END_IF
	
2300: // Clip open Place
	bCylinderCheck := TRUE;
	Clips[iWorkingIndex].M_Retract();
	bCylinderCheck := Clips[iWorkingIndex].InRearPosition AND bCylinderCheck;
	IF bSyncPlace THEN
		Clips[1].M_Retract();
		bCylinderCheck := Clips[1].InRearPosition AND bCylinderCheck;
	END_IF	
	 
	IF bCylinderCheck THEN
		tonTimeOut.IN := FALSE;
		uiExecutingStep:=2400;
	END_IF 
	 tonTimeOut.IN := TRUE;
	IF tonTimeOut.q THEN
		tonTimeOut.IN := FALSE;
		_Abort := TRUE;
		strStatus :='FB_OutRobot_BoxMoveReverse Step 2300: Clip place open timeout';
	END_IF  
	  
2400: // Clip up Placing
	bCylinderCheck := TRUE;
	Cylinders[iWorkingIndex].M_Retract();
	bCylinderCheck := Cylinders[iWorkingIndex].InRearPosition AND bCylinderCheck;
	IF bSyncPlace THEN
		Cylinders[1].M_Retract();
		bCylinderCheck := Cylinders[1].InRearPosition AND bCylinderCheck;
	END_IF	
	 
	IF bCylinderCheck THEN
		tonTimeOut.IN := FALSE;
		uiExecutingStep:=2500;
	END_IF 
	 tonTimeOut.IN := TRUE;
	IF tonTimeOut.q THEN
		tonTimeOut.IN := FALSE;
		_Abort := TRUE;
		strStatus :='FB_OutRobot_BoxMoveReverse Step 2400: Cylinder place up timeout';
	END_IF  
	
2500: // If Next place
	IF iWorkingIndex>=1 OR bSyncPlace OR NOT UseB THEN
		uiExecutingStep:=2600;
		// Finish
	ELSE	
		iWorkingIndex := iWorkingIndex+1;
	  	uiExecutingStep:=2000;
	END_IF

2600: // Move conveyor a bit
		  IF bMotorMoveForward THEN
			 bMoveConveyorForward:=TRUE;//ConveyorMotor.M_MoveForward();
			 bMoveConveyorBackrward:=FALSE;
		  ELSE	 
			  bMoveConveyorForward:=FALSE;
			  bMoveConveyorBackrward:=TRUE;
	 		 ConveyorMotor.M_MoveBackward(); 
		  END_IF
		tonTimeDelay.IN := NOT SensorOnConveyor;		
		IF tonTimeDelay.Q THEN
			uiExecutingStep:=2700;
		END_IF
2700: // Stop movor
		bMoveConveyorForward:=FALSE;
		bMoveConveyorBackrward:=FALSE;
		ConveyorMotor.M_MotorStop();
		tonTimeDelay.IN := FALSE;
		IF ConveyorMotor.InStopped THEN
			uiExecutingStep:=3000;
		END_IF
3000: // Finish	
	_Executed:=TRUE;
	
END_CASE
	
IF NOT Execute THEN
	eState:=STATE_RESETTING;
END_IF
IF _Error THEN
	eState:=STATE_ERROR;
END_IF
IF _Abort THEN
	eSTATE:=STATE_ABORTING;
END_IF
IF _Executed THEN
	eSTATE:=STATE_Done;
END_IF
END_METHOD

